# B&R Automation Studio project Soiled_PLC
Automation Studio 4.10.2.37; technology packages: mapp 5.15.0, mappView 5.15.1

## Configuration DisplayCTT11

CPU , AutomationRuntime S3.09, Build 4.1.2, Vc V4.21.1

### Task classes (Cpu.sw)
```
Cyclic#1 (cycle 10000 us, tolerance 10000 us):
  ClientPane <- Displays.ClientPanel.prg
  Client <- Displays.Client.prg
  zzClientTe <- Displays.zzClientText.prg
Cyclic#4 (cycle 100000 us, tolerance 100000 us):
  zzSQLDrive <- SQL.zzSQLDriver.prg
VcDataObjects: CT11 <- Displays.CT11.dob
Binaries: vcdsint, vcctext, arialbd, verdanab, vcalarm, vcshared, vcpdsw, vccline, vcgclass, vccbtn, vcresman, vccnum, vcchspot, vccstr, vccshape, vcfile, Displa03, vcrt, vcbclass, vcfntttf, verdana, vcdsloc, vccovl, arial, Displa02, vcpfmtcx, visvc, Displa, vcmgr, vctcal, vcptelo, vcpdpp30, vcpfpp30, vcpdvnc, vcnet, Displa01, ashwd, sysconf, asfw, arconfig, iomap
Libraries: DispLib, zzSQL_Lib, AsDb, IecCheck, AsString, sys_lib, Ethernet, AsTCP, Visapi, AsARCfg, AsETH, AsIecCon, standard, runtime, astime, fileio, dataobj
```

### Hardware
```
CTT11 : 4PP420.1043-K37 v1.0.1.3
  Connector IF5:
    ActivateDevice = 1
    Mode = Manual
    InternetAddress = 10.8.4.10
    SubnetMask = 255.255.240.0
    Vnc1
    VncVcObjectName1 = CT11
    VncKeyMappingFile1 = VC\PS2-Keyboard.dis
    VncAuthentication1 = 1
    VncPasswordViewOnly1 = 7701
    VncPasswordViewControl1 = medoc
    VncRefreshRate1 = 500
  PermanentPvSize = 17
  RemanentGlobalPvSize = 4300
  VolatileGlobalPvSize = 150000
  PreservePermanentPvMemory = 1
  RebootPowerfail = 2
  Cyclic1Duration = 10000
  Cyclic1Tolerance = 10000
  Cyclic2Duration = 20000
  Cyclic2Tolerance = 20000
  Cyclic3Duration = 50000
  Cyclic3Tolerance = 50000
  Cyclic4Duration = 100000
  Cyclic4Tolerance = 100000
  Cyclic5Duration = 200000
  Cyclic5Tolerance = 200000
  Cyclic6Duration = 500000
  Cyclic6Tolerance = 500000
  Cyclic7Duration = 1000000
  Cyclic7Tolerance = 1000000
  Cyclic8Duration = 10000
  Cyclic8Tolerance = 30000000
  EthernetDefaultGateway = 10.8.15.254
  VcObjectName = CT11
```

### Cpu.per - CTT11/Cpu.per
```iecst
(********************************************************************
 * COPYRIGHT --
 ********************************************************************
 * File: Cpu.per
 * Author: Dave
 * Created: July 20, 2011
 ********************************************************************
 * Declaration of permanent variables
 ********************************************************************)
VAR_CONFIG
	ClientServerIP AT %M0;
END_VAR
```

## Configuration DisplayPCT04

CPU , AutomationRuntime C4.72, Build 4.1.2, Vc V4.72.0

### Task classes (Cpu.sw)
```
Cyclic#1:
  ClientData <- Displays.ClientDataEntry.prg
  ClientPane <- Displays.ClientPanel.prg
  Client <- Displays.Client.prg
  zzClientTe <- Displays.zzClientText.prg
Cyclic#4:
  zzSQLDrive <- SQL.zzSQLDriver.prg
VcDataObjects: PCT04 <- Displays.PCT04.dob
Binaries: vcrt, vcpk, vcfntttf, verdana, vcctext, arial, verdanab, vccovl, vcpfmtcx, vccbtn, vcdsint, vcpdsw, vcpdpp30, vcshared, vcmgr, vcpfpp30, visvc, vcalarm, vcfile, vccnum, vccstr, vcresman, vcgclass, vcdsloc, arialbd, vcptelo, vctcal, vcchspot, vcbclass, vccline, PCT0402, PCT0401, PCT0403, ashwd, sysconf, asfw, iomap, arconfig, vccbmp, Data1, vccshape, vcnet, Data102, Data103, vcpdvnc, Data101
Libraries: DispLib, standard, asieccon, astime, runtime, IecCheck, AsString, sys_lib, astcp, visapi, zzSQL_Lib, AsDb, dataobj, asarcfg, aseth, fileio
```

### Hardware
```
PCT04 : 4PP065.0571-K05 v1.0.2.2
  Connector IF5:
    ActivateDevice = 1
    Mode = Manual
    InternetAddress = 10.8.4.10
    SubnetMask = 255.255.240.0
    Vnc1
    VncVcObjectName1 = PCT04
    VncKeyMappingFile1 = VC\PS2-Keyboard.dis
    VncAuthentication1 = 1
    VncPasswordViewControl1 = medoc
  ConfigurationID = AS4_7_NorthFleetA5_DisplayPCT04
  PermanentPvSize = 17
  RemanentGlobalPvSize = 4300
  VolatileGlobalPvSize = 150000
  EthernetDefaultGateway = 10.8.15.254
  VcObjectName = PCT04
  KeyMappingFile = 4PP065.0571-K05d.dis
```

## Configuration Supertrack

CPU X20CP1586, AutomationRuntime C4.90, Build 4.1.2, Safety 1.10, Vc V4.72.0

### Task classes (Cpu.sw)
```
Cyclic#1 (cycle 1000 us, tolerance 1000 us):
  4_spn1 <- (binary)
  USB_Pmem <- (binary)
  zzClearMem <- (binary)
  can_dry1 <- (binary)
  zzSQLid <- (binary)
  17_svc2 <- (binary)
  18_svc3 <- (binary)
  20_sic3 <- (binary)
  11_spi1 <- (binary)
  17_sp6 <- (binary)
  8_sp8 <- (binary)
  3_svc2 <- (binary)
  2_svc1 <- (binary)
  9_sp6 <- (binary)
  17_sic1 <- (binary)
  8_svc1 <- (binary)
  50_stnsa1 <- (binary)
Cyclic#2 (cycle 10000 us, tolerance 10000 us):
  zzTC2str <- Sequences.10ms.Scan.zzTC2str.prg
  zzGetTime <- Timestamp.zzGetTime.prg
  zzStd <- Sequences.10ms.zzStd.prg
  zzEditBag <- Sequences.10ms.zzEditBag.prg
  zzForceI <- Sequences.10ms.zzForceI.prg
  zzConst <- Sequences.10ms.zzConst.prg
  zzBagID <- Sequences.10ms.zzBagID.prg
  zzTrip <- Sequences.10ms.zzTrip.prg
  zzStnMix <- Sequences.10ms.zzStnMix.prg
  zzBagShuff <- Sequences.10ms.zzBagShuffle.prg
  zzBITcal <- Sequences.10ms.zzBITcal.prg
  zzStnSer <- Sequences.10ms.zzStnSer.prg
  zzcp10ser <- Sequences.10ms.zzcp10ser.prg
  zzStatus <- Sequences.10ms.zzStatus.prg
  zzCusFIFO <- Sequences.10ms.zzCusFIFO.prg
  0_sbelt <- Sequences.10ms.0_sbelt.prg [disabled]
  50_stns1_7 <- Sequences.10ms.50_stns1_7.prg
  50_stn8_14 <- Sequences.10ms.50_stn8_14.prg
  2_stb1B <- Sequences.10ms.2_stb1.prg
  3_clu_1 <- Sequences.10ms.3_clu_1.prg
  4_pn <- Sequences.10ms.4_pn.prg
  5_pf <- Sequences.10ms.5_pf.prg
  6_sdc1 <- Sequences.10ms.6_sdc1.prg
  7_sdc2 <- Sequences.10ms.7_sdc2.prg
  8_sdc3 <- Sequences.10ms.8_sdc3.prg
  9_sdc4 <- Sequences.10ms.9_sdc4.prg
  10_sdc5 <- Sequences.10ms.10_sdc5.prg
  11_sdc6 <- Sequences.10ms.11_sdc6.prg
  12_sdc7 <- Sequences.10ms.12_sdc7.prg
  13_sdc8 <- Sequences.10ms.13_sdc8.prg
  14_sdc9 <- Sequences.10ms.14_sdc9.prg
  15_cbc1 <- Sequences.10ms.15_cbc1.prg
  16_cic1 <- Sequences.10ms.16_cic1.prg
  17_cic2 <- Sequences.10ms.17_cic2.prg
  18_cic3 <- Sequences.10ms.18_cic3.prg
  19_cic4 <- Sequences.10ms.19_cic4.prg
  20_cp1 <- Sequences.10ms.20_cp17.prg
  21_cpi1 <- Sequences.10ms.21_cpi1.prg
  22_cpi2 <- Sequences.10ms.22_cpi2.prg
  23_cpi3 <- Sequences.10ms.23_cpi3.prg
  24_cpi4 <- Sequences.10ms.24_cpi4.prg
  25_cvc1 <- Sequences.10ms.25_cvc1.prg
  26_cp3 <- Sequences.10ms.26_cp3.prg
  27_cp17 <- Sequences.10ms.27_cp17.prg
  28_cp16 <- Sequences.10ms.28_cp16.prg
  29_cp15 <- Sequences.10ms.29_cp15.prg
  30_cp14 <- Sequences.10ms.30_cp14.prg
  31_cp2 <- Sequences.10ms.31_cp2.prg
  32_clu_2 <- Sequences.10ms.3_clu_2.prg
  33_stb2_A <- Sequences.10ms.32_stb2.prg
  34_cpi5 <- Sequences.10ms.34_cpi5.prg
  35_cic5 <- Sequences.10ms.35_cic5.prg
  36_cic6 <- Sequences.10ms.36_cic6.prg
  37_cpi6 <- Sequences.10ms.37_cpi6.prg
  38_cp10 <- Sequences.10ms.38_cp10.prg
  39_cpc1 <- Sequences.10ms.39_cpc1.prg
  40_cp4 <- Sequences.10ms.40_cp4.prg
  41_cp8 <- Sequences.10ms.41_cp8.prg
  42_cp9 <- Sequences.10ms.42_cp9.prg
  43_cp12 <- Sequences.10ms.43_cp12.prg
  44_cpr2 <- Sequences.10ms.44_cpr2.prg
  45_cpr3 <- Sequences.10ms.45_cpr3.prg
  46_cpr4 <- Sequences.10ms.46_cpr4.prg
  47_cpr1 <- Sequences.10ms.47_cpr1.prg
  48_cp6 <- Sequences.10ms.48_cp6.prg
  ssr <- Sequences.10ms.ssr.prg  // speed reducer before SDC2
  zzUld_4 <- Sequences.10ms.zzUld_4.prg
  zzUld_4a <- Sequences.10ms.zzUld_4a.prg [disabled]
  zzForceO <- Sequences.10ms.zzForceO.prg
  zzIndi <- Sequences.10ms.zzIndi.prg [disabled]
  zzTCPIP <- Sequences.10ms.zzTCPIP.prg
  zzIO <- Sequences.10ms.zzIO.prg
  zzOk <- Sequences.10ms.zzOk.prg
  zzDataStor <- Data_BackUp.zzDataStore.prg
  zzTvText <- SQL.zzTvText.prg
  ServerPane <- Displays.ServerPanel.prg
  Server <- Displays.Server.prg
  zzClientTe <- Displays.zzClientText.prg [disabled]
  zzHttpDriv <- http_Lib.zzHttpDriver.prg [disabled]
  zzGetName1 <- SQL.zzGetNamesSQL.zzGetNameSQL.prg [disabled]
  zzTC2end <- Sequences.10ms.Scan.zzTC2end.prg
Cyclic#3:
  zzGetNames <- Sequences.zzGetNames.prg [disabled]
Cyclic#4:
  SafetyUI <- Safety.SafetyUI.prg [disabled]
Cyclic#5:
  HoistServe <- HoistLibrary.HoistServer.prg
  AccessCont <- Safety.AccessControl.prg
  Safety <- Safety.Safety.prg [disabled]
  can_drv1 <- Sequences.200ms.CAN.can_drv1.prg
  can_drv2 <- Sequences.200ms.CAN.can_drv2.prg
  zzWeigh <- Sequences.200ms.zzWeigh.prg
  zzAlarms <- Sequences.200ms.zzAlarms.prg
  zzReport <- Sequences.200ms.Reports.zzReport.prg
  zzStn_Q <- Sequences.200ms.zzStn_Q.prg
  zzTime <- Sequences.200ms.zzTime.prg  // System running time
  CAN_Live <- Sequences.200ms.CAN.CAN_Live.prg
  httpServer <- http_Lib.httpServer.prg [disabled]
Cyclic#8:
  zzModuleLo <- CustomLogs.zzModuleLog.prg
  zzSQLDrive <- SQL.zzSQLDriver.prg [disabled]
  zzWeighSta <- CustomLogs.zzWeighStatus.prg [disabled]
DataObjects: can2_cmd <- Sequences.200ms.CAN.can2_cmd.dob, can1_cmd <- Sequences.200ms.CAN.can1_cmd.dob, arsdmsvp, arsdmhtm, arsdmsvg
Binaries: TCData, udbdef, mvLoader, FWRules, TCLang, iomap, asfw, arconfig, ashwd, sysconf, Role, User, ashwac, TC, OpcUaMap, vcfntttf, vcfile, vcshared, vccshape, vcgclass, arial, CT1102, vcchspot, vcdsint, PCT0403, vccbtn, vcdsloc, vccovl, vccline, vcctext, vcalarm, vcbclass, vcrt, vccnum, vccstr, CT1103, arialbd, PCT0402, vcpdsw, verdanab, verdana, webserv, arsdm
Libraries: ABB_EPL, AsEPL, AsBrMath, AsIOAcc, AsSafety, MTBasics, MTTypes, Ldg_Funct, FileMgr, KanLinkLib, OPCuA, FC302, DataBackUp, standard, runtime, FileIO, Ethernet, dvframe, DataObj, OPERATOR, CAN_Lib, AsTime, AsString, SupLib4, sys_lib, AsTCP, KGstring, AsETH, AsBrStr, AsBrWStr, AsUSB, AsMem, AsArLog, AsUDP, brsystem, AsIODiag, AsARCfg, AsIecCon, IecCheck, AsPciStr, DispLib, zzSQL_Lib, AsDb, KGstdLib, mnParamLib, KL_UserLib, AsHttp, SUP, asxml, ascanopen, arssl, SupFile, vcresman, WETCAN2
```

### Hardware
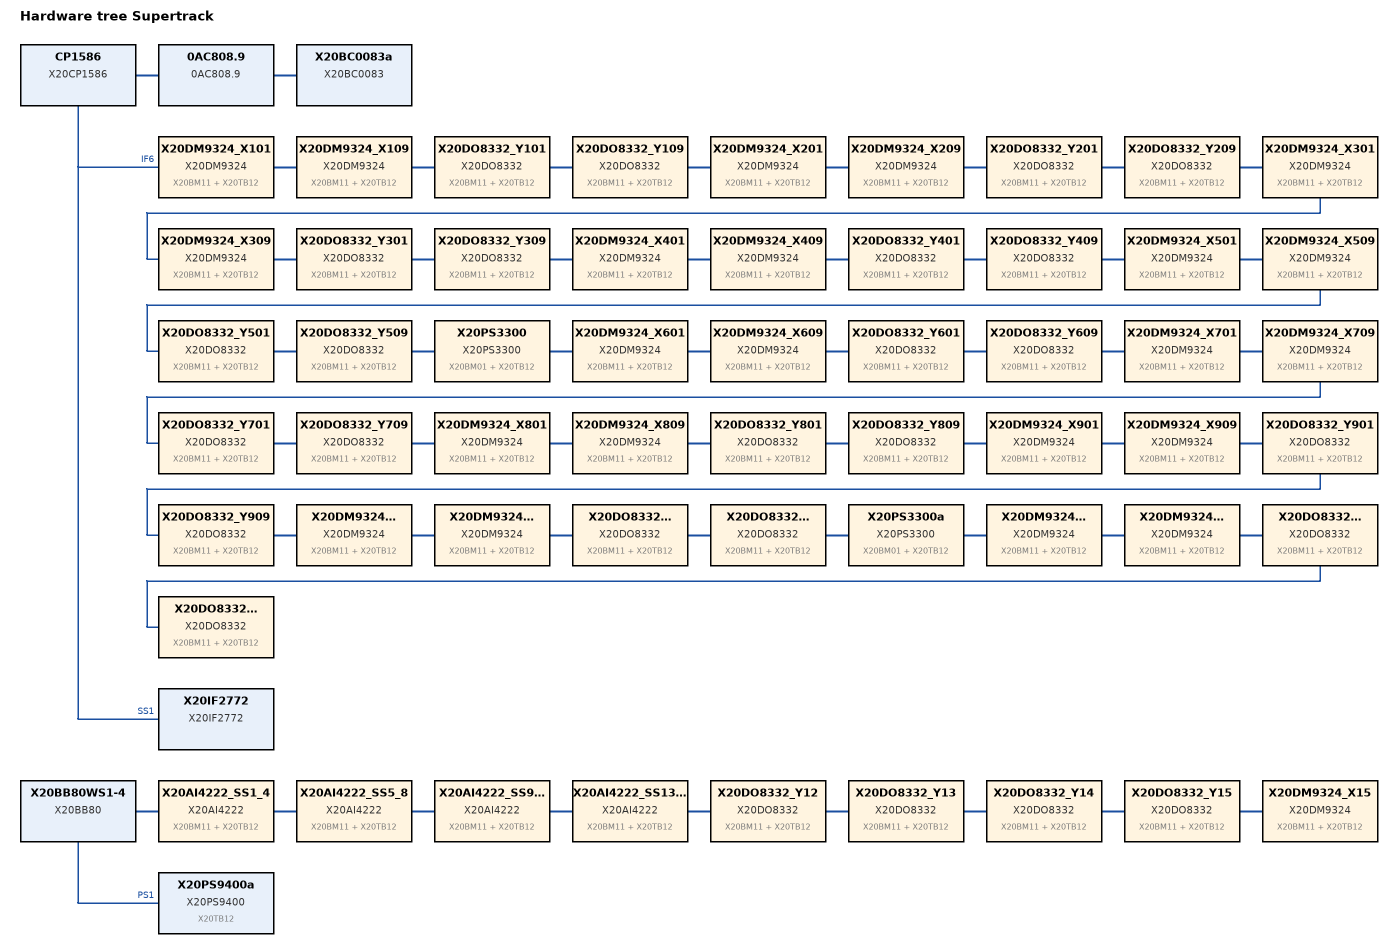
```
0AC808.9 : 0AC808.9 v1.0.0.0  [ETH1 -> CP1586.IF3 [Cable Type=PowerlinkCable, Length=10, Version=1.0.0.3]; ETH8 -> X20BC0083a.PLK1 [Cable Type=PowerlinkCable, Length=10, Version=1.0.0.3]]
CP1586 : X20CP1586 v1.9.0.0
  Connector IF2:
    ActivateDevice = 1
    Baudrate = 100
    Mode = Manual
    InternetAddress = 10.8.4.20
  ConfigurationID = AS4_2_BaseStandard_Supertrack
  UserRamSize = 200000
  RemMemSize = 200000
  PermanentPvSize = 47756
  RemanentGlobalPvSize = 5000
  VolatileGlobalPvSize = 900000
  ClearNvMemoryAfterShutdownFlushError = 0
  CyclicFlushRemMemSelector = 1
  EnableUsbRemoteInstall = 1
  EnableCfRemoteInstall = 1
  Cyclic1Duration = 1000
  Cyclic1Tolerance = 1000
  Cyclic2Duration = 10000
  Cyclic2Tolerance = 10000
  FileDevice1
  FileDeviceName1 = USBStick
  FileDevicePath1 = /bd0\
  ActivateDaylightSavingTime = 1
  ActivateSntp = 1
  SntpcServAddr1 = 10.8.15.254
  EthernetHostName = SupertrackPLC
  EthernetDefaultGateway = 10.8.15.254
  FtpUser1
  FtpUsername1 = admin
  FtpUserPassword1 = vwQCGOhDKwuFhUdMhisKVJgiKzmoNTQazzJQnTTJsZU=  // admin
  FtpUserSalt1 = XFuy8Eo/
  FTPAccessRight1 = 0
  ActivateOpcUa = 1
  OpcUa_AuthenticationTokenType_EnableAnonymous = 0
  OpcUaInformationModels_PV_Version = 1
X20AI4222_SS13_14 : X20AI4222 v1.1.0.0  [SS1 -> X20TB12aq.SS; SL -> X20BM11am.SL1]
  Supervision = off
X20AI4222_SS1_4 : X20AI4222 v1.1.0.0  [SS1 -> X20TB12as.SS; SL -> X20BM11ak.SL1]
  Supervision = off
X20AI4222_SS5_8 : X20AI4222 v1.1.0.0  [SS1 -> X20TB12n.SS; SL -> X20BM11ao.SL1]
  Supervision = off
X20AI4222_SS9_12 : X20AI4222 v1.1.0.0  [SS1 -> X20TB12aw.SS; SL -> X20BM11av.SL1]
  Supervision = off
X20BB80WS1-4 : X20BB80 v1.1.0.0
X20BC0083a : X20BC0083 v2.14.0.0  [PLK1 -> 0AC808.9.ETH8 (NodeNumber=2) [Cable Type=PowerlinkCable, Length=10, Version=1.0.0.3]; SL -> X20BB80WS1-4.SL1]
  Supervision = off
X20BM01 : X20BM01 v2.2.0.0  [X2X1 -> X20BM11s.X2X2]
X20BM01a : X20BM01 v2.2.0.0  [X2X1 -> X20BM11aj.X2X2]
X20BM11 : X20BM11 v1.1.0.0  [X2X1 -> CP1586.IF6]
X20BM11a : X20BM11 v1.1.0.0  [X2X1 -> X20BM11.X2X2]
X20BM11aa : X20BM11 v1.1.0.0  [X2X1 -> X20BM11z.X2X2]
X20BM11ab : X20BM11 v1.1.0.0  [X2X1 -> X20BM11aa.X2X2]
X20BM11ac : X20BM11 v1.1.0.0  [X2X1 -> X20BM11ab.X2X2]
X20BM11ad : X20BM11 v1.1.0.0  [X2X1 -> X20BM11ac.X2X2]
X20BM11ae : X20BM11 v1.1.0.0  [X2X1 -> X20BM11ad.X2X2]
X20BM11af : X20BM11 v1.1.0.0  [X2X1 -> X20BM11ag.X2X2]
X20BM11ag : X20BM11 v1.1.0.0  [X2X1 -> X20BM11as.X2X2]
X20BM11ah : X20BM11 v1.1.0.0  [X2X1 -> X20BM11at.X2X2]
X20BM11ai : X20BM11 v1.1.0.0  [X2X1 -> X20BM11au.X2X2]
X20BM11aj : X20BM11 v1.1.0.0  [X2X1 -> X20BM11ai.X2X2]
X20BM11ak : X20BM11 v1.1.0.0  [X2X1 -> X20BB80WS1-4.IF1]
X20BM11al : X20BM11 v1.1.0.0  [X2X1 -> X20BM11an.X2X2]
X20BM11am : X20BM11 v1.1.0.0  [X2X1 -> X20BM11av.X2X2]
X20BM11an : X20BM11 v1.1.0.0  [X2X1 -> X20BM11bc.X2X2]
X20BM11ao : X20BM11 v1.1.0.0  [X2X1 -> X20BM11ak.X2X2]
X20BM11as : X20BM11 v1.1.0.0  [X2X1 -> X20BM11ae.X2X2]
X20BM11at : X20BM11 v1.1.0.0  [X2X1 -> X20BM11af.X2X2]
X20BM11au : X20BM11 v1.1.0.0  [X2X1 -> X20BM11ah.X2X2]
X20BM11av : X20BM11 v1.1.0.0  [X2X1 -> X20BM11ao.X2X2]
X20BM11aw : X20BM11 v1.1.0.0  [X2X1 -> X20BM11am.X2X2]
X20BM11ax : X20BM11 v1.1.0.0  [X2X1 -> X20BM01a.X2X2]
X20BM11ay : X20BM11 v1.1.0.0  [X2X1 -> X20BM11ax.X2X2]
X20BM11az : X20BM11 v1.1.0.0  [X2X1 -> X20BM11ay.X2X2]
X20BM11b : X20BM11 v1.1.0.0  [X2X1 -> X20BM11a.X2X2]
X20BM11ba : X20BM11 v1.1.0.0  [X2X1 -> X20BM11az.X2X2]
X20BM11bb : X20BM11 v1.1.0.0  [X2X1 -> X20BM11aw.X2X2]
X20BM11bc : X20BM11 v1.1.0.0  [X2X1 -> X20BM11bb.X2X2]
X20BM11c : X20BM11 v1.1.0.0  [X2X1 -> X20BM11b.X2X2]
X20BM11d : X20BM11 v1.1.0.0  [X2X1 -> X20BM11c.X2X2]
X20BM11e : X20BM11 v1.1.0.0  [X2X1 -> X20BM11d.X2X2]
X20BM11f : X20BM11 v1.1.0.0  [X2X1 -> X20BM11e.X2X2]
X20BM11g : X20BM11 v1.1.0.0  [X2X1 -> X20BM11f.X2X2]
X20BM11h : X20BM11 v1.1.0.0  [X2X1 -> X20BM11g.X2X2]
X20BM11i : X20BM11 v1.1.0.0  [X2X1 -> X20BM11h.X2X2]
X20BM11j : X20BM11 v1.1.0.0  [X2X1 -> X20BM11i.X2X2]
X20BM11k : X20BM11 v1.1.0.0  [X2X1 -> X20BM11j.X2X2]
X20BM11l : X20BM11 v1.1.0.0  [X2X1 -> X20BM11k.X2X2]
X20BM11m : X20BM11 v1.1.0.0  [X2X1 -> X20BM11l.X2X2]
X20BM11n : X20BM11 v1.1.0.0  [X2X1 -> X20BM11m.X2X2]
X20BM11o : X20BM11 v1.1.0.0  [X2X1 -> X20BM11n.X2X2]
X20BM11p : X20BM11 v1.1.0.0  [X2X1 -> X20BM11o.X2X2]
X20BM11q : X20BM11 v1.1.0.0  [X2X1 -> X20BM11p.X2X2]
X20BM11r : X20BM11 v1.1.0.0  [X2X1 -> X20BM11q.X2X2]
X20BM11s : X20BM11 v1.1.0.0  [X2X1 -> X20BM11r.X2X2]
X20BM11t : X20BM11 v1.1.0.0  [X2X1 -> X20BM01.X2X2]
X20BM11u : X20BM11 v1.1.0.0  [X2X1 -> X20BM11t.X2X2]
X20BM11v : X20BM11 v1.1.0.0  [X2X1 -> X20BM11u.X2X2]
X20BM11w : X20BM11 v1.1.0.0  [X2X1 -> X20BM11v.X2X2]
X20BM11x : X20BM11 v1.1.0.0  [X2X1 -> X20BM11w.X2X2]
X20BM11y : X20BM11 v1.1.0.0  [X2X1 -> X20BM11x.X2X2]
X20BM11z : X20BM11 v1.1.0.0  [X2X1 -> X20BM11y.X2X2]
X20DM9324_X1001 : X20DM9324 v1.2.0.0  [SS1 -> X20TB12ak.SS; SL -> X20BM11ah.SL1]
  Supervision = off
X20DM9324_X1009 : X20DM9324 v1.2.0.0  [SS1 -> X20TB12ba.SS; SL -> X20BM11au.SL1]
  Supervision = off
X20DM9324_X101 : X20DM9324 v1.2.0.0  [SS1 -> X20TB12.SS; SL -> X20BM11.SL1]
  Supervision = off
X20DM9324_X109 : X20DM9324 v1.2.0.0  [SS1 -> X20TB12a.SS; SL -> X20BM11a.SL1]
  Supervision = off
X20DM9324_X1101 : X20DM9324 v1.2.0.0  [SS1 -> X20TB12bd.SS; SL -> X20BM11ax.SL1]
  Supervision = off
X20DM9324_X1109 : X20DM9324 v1.2.0.0  [SS1 -> X20TB12be.SS; SL -> X20BM11ay.SL1]
  Supervision = off
X20DM9324_X15 : X20DM9324 v1.2.0.0  [SS1 -> X20TB12ap.SS; SL -> X20BM11al.SL1]
  Supervision = off
X20DM9324_X201 : X20DM9324 v1.2.0.0  [SS1 -> X20TB12d.SS; SL -> X20BM11d.SL1]
  Supervision = off
X20DM9324_X209 : X20DM9324 v1.2.0.0  [SS1 -> X20TB12e.SS; SL -> X20BM11e.SL1]
  Supervision = off
X20DM9324_X301 : X20DM9324 v1.2.0.0  [SS1 -> X20TB12h.SS; SL -> X20BM11h.SL1]
  Supervision = off
X20DM9324_X309 : X20DM9324 v1.2.0.0  [SS1 -> X20TB12i.SS; SL -> X20BM11i.SL1]
  Supervision = off
X20DM9324_X401 : X20DM9324 v1.2.0.0  [SS1 -> X20TB12l.SS; SL -> X20BM11l.SL1]
  Supervision = off
X20DM9324_X409 : X20DM9324 v1.2.0.0  [SS1 -> X20TB12m.SS; SL -> X20BM11m.SL1]
  Supervision = off
X20DM9324_X501 : X20DM9324 v1.2.0.0  [SS1 -> X20TB12q.SS; SL -> X20BM11p.SL1]
  Supervision = off
X20DM9324_X509 : X20DM9324 v1.2.0.0  [SS1 -> X20TB12r.SS; SL -> X20BM11q.SL1]
  Supervision = off
X20DM9324_X601 : X20DM9324 v1.2.0.0  [SS1 -> X20TB12v.SS; SL -> X20BM11t.SL1]
  Supervision = off
X20DM9324_X609 : X20DM9324 v1.2.0.0  [SS1 -> X20TB12w.SS; SL -> X20BM11u.SL1]
  Supervision = off
X20DM9324_X701 : X20DM9324 v1.2.0.0  [SS1 -> X20TB12z.SS; SL -> X20BM11x.SL1]
  Supervision = off
X20DM9324_X709 : X20DM9324 v1.2.0.0  [SS1 -> X20TB12aa.SS; SL -> X20BM11y.SL1]
  Supervision = off
X20DM9324_X801 : X20DM9324 v1.2.0.0  [SS1 -> X20TB12ad.SS; SL -> X20BM11ab.SL1]
  Supervision = off
X20DM9324_X809 : X20DM9324 v1.2.0.0  [SS1 -> X20TB12ae.SS; SL -> X20BM11ac.SL1]
  Supervision = off
X20DM9324_X901 : X20DM9324 v1.2.0.0  [SS1 -> X20TB12ah.SS; SL -> X20BM11as.SL1]
  Supervision = off
X20DM9324_X909 : X20DM9324 v1.2.0.0  [SS1 -> X20TB12aj.SS; SL -> X20BM11ag.SL1]
  Supervision = off
X20DO8332_Y1001 : X20DO8332 v1.5.0.0  [SS1 -> X20TB12al.SS; SL -> X20BM11ai.SL1]
  Supervision = off
X20DO8332_Y1009 : X20DO8332 v1.5.0.0  [SS1 -> X20TB12am.SS; SL -> X20BM11aj.SL1]
  Supervision = off
X20DO8332_Y101 : X20DO8332 v1.5.0.0  [SS1 -> X20TB12b.SS; SL -> X20BM11b.SL1]
  Supervision = off
X20DO8332_Y109 : X20DO8332 v1.5.0.0  [SS1 -> X20TB12c.SS; SL -> X20BM11c.SL1]
  Supervision = off
X20DO8332_Y1101 : X20DO8332 v1.5.0.0  [SS1 -> X20TB12bf.SS; SL -> X20BM11az.SL1]
  Supervision = off
X20DO8332_Y1109 : X20DO8332 v1.5.0.0  [SS1 -> X20TB12bg.SS; SL -> X20BM11ba.SL1]
  Supervision = off
X20DO8332_Y12 : X20DO8332 v1.5.0.0  [SS1 -> X20TB12bb.SS; SL -> X20BM11aw.SL1]
  Supervision = off
X20DO8332_Y13 : X20DO8332 v1.5.0.0  [SS1 -> X20TB12bc.SS; SL -> X20BM11bb.SL1]
  Supervision = off
X20DO8332_Y14 : X20DO8332 v1.5.0.0  [SS1 -> X20TB12bh.SS; SL -> X20BM11bc.SL1]
  Supervision = off
X20DO8332_Y15 : X20DO8332 v1.5.0.0  [SS1 -> X20TB12ar.SS; SL -> X20BM11an.SL1]
  Supervision = off
X20DO8332_Y201 : X20DO8332 v1.5.0.0  [SS1 -> X20TB12f.SS; SL -> X20BM11f.SL1]
  Supervision = off
X20DO8332_Y209 : X20DO8332 v1.5.0.0  [SS1 -> X20TB12g.SS; SL -> X20BM11g.SL1]
  Supervision = off
X20DO8332_Y301 : X20DO8332 v1.5.0.0  [SS1 -> X20TB12j.SS; SL -> X20BM11j.SL1]
  Supervision = off
X20DO8332_Y309 : X20DO8332 v1.5.0.0  [SS1 -> X20TB12k.SS; SL -> X20BM11k.SL1]
  Supervision = off
X20DO8332_Y401 : X20DO8332 v1.5.0.0  [SS1 -> X20TB12o.SS; SL -> X20BM11n.SL1]
  Supervision = off
X20DO8332_Y409 : X20DO8332 v1.5.0.0  [SS1 -> X20TB12p.SS; SL -> X20BM11o.SL1]
  Supervision = off
X20DO8332_Y501 : X20DO8332 v1.5.0.0  [SS1 -> X20TB12s.SS; SL -> X20BM11r.SL1]
  Supervision = off
X20DO8332_Y509 : X20DO8332 v1.5.0.0  [SS1 -> X20TB12t.SS; SL -> X20BM11s.SL1]
  Supervision = off
X20DO8332_Y601 : X20DO8332 v1.5.0.0  [SS1 -> X20TB12x.SS; SL -> X20BM11v.SL1]
  Supervision = off
X20DO8332_Y609 : X20DO8332 v1.5.0.0  [SS1 -> X20TB12y.SS; SL -> X20BM11w.SL1]
  Supervision = off
X20DO8332_Y701 : X20DO8332 v1.5.0.0  [SS1 -> X20TB12ab.SS; SL -> X20BM11z.SL1]
  Supervision = off
X20DO8332_Y709 : X20DO8332 v1.5.0.0  [SS1 -> X20TB12ac.SS; SL -> X20BM11aa.SL1]
  Supervision = off
X20DO8332_Y801 : X20DO8332 v1.5.0.0  [SS1 -> X20TB12af.SS; SL -> X20BM11ad.SL1]
  Supervision = off
X20DO8332_Y809 : X20DO8332 v1.5.0.0  [SS1 -> X20TB12ag.SS; SL -> X20BM11ae.SL1]
  Supervision = off
X20DO8332_Y901 : X20DO8332 v1.5.0.0  [SS1 -> X20TB12ai.SS; SL -> X20BM11af.SL1]
  Supervision = off
X20DO8332_Y909 : X20DO8332 v1.5.0.0  [SS1 -> X20TB12az.SS; SL -> X20BM11at.SL1]
  Supervision = off
X20IF2772 : X20IF2772 v1.5.0.0  [SS -> CP1586.SS1]
X20PS3300 : X20PS3300 v1.3.0.0  [SS1 -> X20TB12u.SS; SL -> X20BM01.SL1]
  Supervision = off
X20PS3300a : X20PS3300 v1.3.0.0  [SS1 -> X20TB12an.SS; SL -> X20BM01a.SL1]
  Supervision = off
X20PS9400a : X20PS9400 v1.7.0.0  [SS1 -> X20TB12ao.SS; PS -> X20BB80WS1-4.PS1]
  Supervision = off
X20TB12 : X20TB12 v1.0.0.0
X20TB12a : X20TB12 v1.0.0.0
X20TB12aa : X20TB12 v1.0.0.0
X20TB12ab : X20TB12 v1.0.0.0
X20TB12ac : X20TB12 v1.0.0.0
X20TB12ad : X20TB12 v1.0.0.0
X20TB12ae : X20TB12 v1.0.0.0
X20TB12af : X20TB12 v1.0.0.0
X20TB12ag : X20TB12 v1.0.0.0
X20TB12ah : X20TB12 v1.0.0.0
X20TB12ai : X20TB12 v1.0.0.0
X20TB12aj : X20TB12 v1.0.0.0
X20TB12ak : X20TB12 v1.0.0.0
X20TB12al : X20TB12 v1.0.0.0
X20TB12am : X20TB12 v1.0.0.0
X20TB12an : X20TB12 v1.0.0.0
X20TB12ao : X20TB12 v1.0.0.0
X20TB12ap : X20TB12 v1.0.0.0
X20TB12aq : X20TB12 v1.0.0.0
X20TB12ar : X20TB12 v1.0.0.0
X20TB12as : X20TB12 v1.0.0.0
X20TB12aw : X20TB12 v1.0.0.0
X20TB12az : X20TB12 v1.0.0.0
X20TB12b : X20TB12 v1.0.0.0
X20TB12ba : X20TB12 v1.0.0.0
X20TB12bb : X20TB12 v1.0.0.0
X20TB12bc : X20TB12 v1.0.0.0
X20TB12bd : X20TB12 v1.0.0.0
X20TB12be : X20TB12 v1.0.0.0
X20TB12bf : X20TB12 v1.0.0.0
X20TB12bg : X20TB12 v1.0.0.0
X20TB12bh : X20TB12 v1.0.0.0
X20TB12c : X20TB12 v1.0.0.0
X20TB12d : X20TB12 v1.0.0.0
X20TB12e : X20TB12 v1.0.0.0
X20TB12f : X20TB12 v1.0.0.0
X20TB12g : X20TB12 v1.0.0.0
X20TB12h : X20TB12 v1.0.0.0
X20TB12i : X20TB12 v1.0.0.0
X20TB12j : X20TB12 v1.0.0.0
X20TB12k : X20TB12 v1.0.0.0
X20TB12l : X20TB12 v1.0.0.0
X20TB12m : X20TB12 v1.0.0.0
X20TB12n : X20TB12 v1.0.0.0
X20TB12o : X20TB12 v1.0.0.0
X20TB12p : X20TB12 v1.0.0.0
X20TB12q : X20TB12 v1.0.0.0
X20TB12r : X20TB12 v1.0.0.0
X20TB12s : X20TB12 v1.0.0.0
X20TB12t : X20TB12 v1.0.0.0
X20TB12u : X20TB12 v1.0.0.0
X20TB12v : X20TB12 v1.0.0.0
X20TB12w : X20TB12 v1.0.0.0
X20TB12x : X20TB12 v1.0.0.0
X20TB12y : X20TB12 v1.0.0.0
X20TB12z : X20TB12 v1.0.0.0
```

### 230104.iom - CP1586/230104.iom
```iecst
08:04:57, Error= -2147217873,  CmdExport  [Microsoft][ODBC Microsoft Access Driver] The changes you requested to the table were not successful because they would create duplicate values in the index, primary key, or relationship.  Change the data in the field or fields that contain duplicate data, remove the index, or redefine the index to permit duplicate entries and try again.
```

### 230121.iom - CP1586/230121.iom
```iecst
16:15:44, Error= -2147217873,  CmdExport  [Microsoft][ODBC Microsoft Access Driver] The changes you requested to the table were not successful because they would create duplicate values in the index, primary key, or relationship.  Change the data in the field or fields that contain duplicate data, remove the index, or redefine the index to permit duplicate entries and try again.
```

### Cpu.per - CP1586/Cpu.per
```iecst
(********************************************************************
 * COPYRIGHT --
 ********************************************************************
 * File: Cpu.per
 * Author: Dave
 * Created: November 19, 2010
 ********************************************************************
 * Declaration of permanent variables
 ********************************************************************)
VAR_CONFIG
	C AT %MW0; (* *)
	D AT %MW200; (* *)
	D32 AT %MD16200; (* *)
	RB_Posn AT %M20200; (* *)
	RB_Perm AT %M22632; (* *)
	SQL AT %M22696; (* *)
	ReportBuffer AT %M22956; (* *)
	Bag AT %M31756; (* *)
END_VAR
```

### IoMap.iom - CP1586/IoMap.iom
```iecst
(********************************************************************
 * COPYRIGHT --
 ********************************************************************
 * File: IoMap.iom
 * Author: Dave
 * Created: November 19, 2010
 ********************************************************************
 * IO mapping file
 ********************************************************************)
VAR_CONFIG
	OK[1] AT %IX."X20DM9324_X101".ModuleOk;
	X[1].X01 AT %IX."X20DM9324_X101".DigitalInput01; (*CDC 5 Bag at buffer   *)
	X[1].X02 AT %IX."X20DM9324_X101".DigitalInput02; (*CDC 5 Bag at buffer stop *)
	X[1].X03 AT %IX."X20DM9324_X101".DigitalInput03; (*CDC 5 Bag in discharger*)
	X[1].X04 AT %IX."X20DM9324_X101".DigitalInput04; (*CDC 5 Bag out of discharger *)
	X[1].X05 AT %IX."X20DM9324_X101".DigitalInput05; (*CDC 5 Drop load *)
	X[1].X06 AT %IX."X20DM9324_X101".DigitalInput06; (*CDC 5 Load dropped *)
	X[1].X07 AT %IX."X20DM9324_X101".DigitalInput07; (*CDC 6 Bag at buffer *)
	X[1].X08 AT %IX."X20DM9324_X101".DigitalInput08; (*CDC 6 Bag at buffer stop *)
	OK[2] AT %IX."X20DM9324_X109".ModuleOk;
	X[1].X09 AT %IX."X20DM9324_X109".DigitalInput01; (*CDC 6 Bag in discharger  *)
	X[1].X10 AT %IX."X20DM9324_X109".DigitalInput02; (*CDC 6 Bag out of discharger *)
	X[1].X11 AT %IX."X20DM9324_X109".DigitalInput03; (*CDC 6 Drop load *)
	X[1].X12 AT %IX."X20DM9324_X109".DigitalInput04; (*CDC 6 Load dropped  *)
	X[1].X13 AT %IX."X20DM9324_X109".DigitalInput05; (*CDC 7 Bag at buffer  *)
	X[1].X14 AT %IX."X20DM9324_X109".DigitalInput06; (*CDC 7 Bag at buffer stop *)
	X[1].X15 AT %IX."X20DM9324_X109".DigitalInput07; (*CDC 7 Bag in discharger *)
	X[1].X16 AT %IX."X20DM9324_X109".DigitalInput08; (*CDC 7 Bag out of discharger  *)
	OK[3] AT %IX."X20DO8332_Y101".ModuleOk;
	Y[1].Y01 AT %QX."X20DO8332_Y101".DigitalOutput01; (*CP 10 Select point to SDC 5 *)
	Y[1].Y02 AT %QX."X20DO8332_Y101".DigitalOutput02; (*CDC 5 Open buffer stop *)
	Y[1].Y03 AT %QX."X20DO8332_Y101".DigitalOutput03; (*CDC 5 Open discharger stop *)
	Y[1].Y04 AT %QX."X20DO8332_Y101".DigitalOutput04; (*CDC 5 Steady cylinders *)
	Y[1].Y05 AT %QX."X20DO8332_Y101".DigitalOutput05; (*CDC 5 Bag ready *)
	Y[1].Y06 AT %QX."X20DO8332_Y101".DigitalOutput06; (*CDC 5 Open bag *)
	Y[1].Y07 AT %QX."X20DO8332_Y101".DigitalOutput07; (*CP 11 Select point to SDC 6 *)
	Y[1].Y08 AT %QX."X20DO8332_Y101".DigitalOutput08; (*CDC 6 Open buffer stop *)
	OK[4] AT %IX."X20DO8332_Y109".ModuleOk;
	Y[1].Y09 AT %QX."X20DO8332_Y109".DigitalOutput01; (*CDC 6 Open discharger stop + CP 14*)
	Y[1].Y10 AT %QX."X20DO8332_Y109".DigitalOutput02; (*CDC 6 Steady cylinders*)
	Y[1].Y11 AT %QX."X20DO8332_Y109".DigitalOutput03; (*CDC 6 Bag ready *)
	Y[1].Y12 AT %QX."X20DO8332_Y109".DigitalOutput04; (*CDC 6 Open bag*)
	Y[1].Y13 AT %QX."X20DO8332_Y109".DigitalOutput05; (*CP 12 Select point to SDC 7 *)
	Y[1].Y14 AT %QX."X20DO8332_Y109".DigitalOutput06; (*CDC 7 Open buffer stop *)
	Y[1].Y15 AT %QX."X20DO8332_Y109".DigitalOutput07; (*CDC 7 Open discharger stop + CP 15*)
	Y[1].Y16 AT %QX."X20DO8332_Y109".DigitalOutput08; (*CDC 7 Steady cylinders *)
	OK[5] AT %IX."X20DM9324_X201".ModuleOk;
	X[2].X01 AT %IX."X20DM9324_X201".DigitalInput01; (*CDC 7 Drop load    *)
	X[2].X02 AT %IX."X20DM9324_X201".DigitalInput02; (*CDC 7 Load dropped *)
	X[2].X03 AT %IX."X20DM9324_X201".DigitalInput03; (*CDC 8 Bag at buffer *)
	X[2].X04 AT %IX."X20DM9324_X201".DigitalInput04; (*CDC 8 Bag at buffer stop *)
	X[2].X05 AT %IX."X20DM9324_X201".DigitalInput05; (*CDC 8 Bag in discharger *)
	X[2].X06 AT %IX."X20DM9324_X201".DigitalInput06; (*CDC 8 Bag out of discharger*)
	X[2].X07 AT %IX."X20DM9324_X201".DigitalInput07; (*CDC 8 Drop load *)
	X[2].X08 AT %IX."X20DM9324_X201".DigitalInput08; (*CDC 8 Load dropped *)
	OK[6] AT %IX."X20DM9324_X209".ModuleOk;
	X[2].X09 AT %IX."X20DM9324_X209".DigitalInput01; (*CDC9 Bag at buffer*)
	X[2].X10 AT %IX."X20DM9324_X209".DigitalInput02; (*CDC 9 Bag at buffer stop *)
	X[2].X11 AT %IX."X20DM9324_X209".DigitalInput03; (*CDC 9 Bag in discharger *)
	X[2].X12 AT %IX."X20DM9324_X209".DigitalInput04; (*CDC 9 Bag out of discharger *)
	X[2].X13 AT %IX."X20DM9324_X209".DigitalInput05; (*CDC 9 Drop load *)
	X[2].X14 AT %IX."X20DM9324_X209".DigitalInput06; (*CDC 9 Load dropped *)
	X[2].X15 AT %IX."X20DM9324_X209".DigitalInput07; (*Spare *)
	X[2].X16 AT %IX."X20DM9324_X209".DigitalInput08; (*CIC 6 Bag at buffer stop *)
	OK[7] AT %IX."X20DO8332_Y201".ModuleOk;
	Y[2].Y01 AT %QX."X20DO8332_Y201".DigitalOutput01; (*CDC 7 Bag ready*)
	Y[2].Y02 AT %QX."X20DO8332_Y201".DigitalOutput02; (*CDC 7 Open bag*)
	Y[2].Y03 AT %QX."X20DO8332_Y201".DigitalOutput03; (*CP13 Select CDC8*)
	Y[2].Y04 AT %QX."X20DO8332_Y201".DigitalOutput04; (*CDC 8 Open buffer stop*)
	Y[2].Y05 AT %QX."X20DO8332_Y201".DigitalOutput05; (*CDC 8 Open discharger stop + CP 16*)
	Y[2].Y06 AT %QX."X20DO8332_Y201".DigitalOutput06; (*CDC 8 Steady cylinders *)
	Y[2].Y07 AT %QX."X20DO8332_Y201".DigitalOutput07; (*CDC 8 Bag ready*)
	Y[2].Y08 AT %QX."X20DO8332_Y201".DigitalOutput08; (*CDC 8 Open bag*)
	OK[8] AT %IX."X20DO8332_Y209".ModuleOk;
	Y[2].Y09 AT %QX."X20DO8332_Y209".DigitalOutput01; (*Spare*)
	Y[2].Y10 AT %QX."X20DO8332_Y209".DigitalOutput02; (*CDC 9 Open buffer stop*)
	Y[2].Y11 AT %QX."X20DO8332_Y209".DigitalOutput03; (*CDC 9 Open discharger stop + CP 17*)
	Y[2].Y12 AT %QX."X20DO8332_Y209".DigitalOutput04; (*CDC 9 Steady cylinders*)
	Y[2].Y13 AT %QX."X20DO8332_Y209".DigitalOutput05; (*CDC 9 Bag ready*)
	Y[2].Y14 AT %QX."X20DO8332_Y209".DigitalOutput06; (*CDC 9 Open bag*)
	Y[2].Y15 AT %QX."X20DO8332_Y209".DigitalOutput07; (*CIC 5 Open buffer stop*)
	Y[2].Y16 AT %QX."X20DO8332_Y209".DigitalOutput08; (*CIC 6 Open buffer stop*)
	OK[9] AT %IX."X20DM9324_X301".ModuleOk;
	X[3].X01 AT %IX."X20DM9324_X301".DigitalInput01; (*Alarm Cancel *)
	X[3].X02 AT %IX."X20DM9324_X301".DigitalInput02; (*Sorting belt A photocell*)
	X[3].X03 AT %IX."X20DM9324_X301".DigitalInput03; (*CLU1 Bag at buffer stop*)
	X[3].X04 AT %IX."X20DM9324_X301".DigitalInput04; (*CLU1 Bag passed stop*)
	X[3].X05 AT %IX."X20DM9324_X301".DigitalInput05; (*CLU1 Bag at loading unit stop*)
	X[3].X06 AT %IX."X20DM9324_X301".DigitalInput06; (*CLU 1 Bag out of loading unit*)
	X[3].X07 AT %IX."X20DM9324_X301".DigitalInput07; (*Sorting belt B photocell*)
	X[3].X08 AT %IX."X20DM9324_X301".DigitalInput08; (*CLU2 Bag at buffer stop*)
	OK[10] AT %IX."X20DM9324_X309".ModuleOk;
	X[3].X09 AT %IX."X20DM9324_X309".DigitalInput01; (*CLU2 Bag passed stop*)
	X[3].X10 AT %IX."X20DM9324_X309".DigitalInput02; (*CLU2 Bag at loading unit stop*)
	X[3].X11 AT %IX."X20DM9324_X309".DigitalInput03; (*CLU2 Bag out of loading unit*)
	X[3].X12 AT %IX."X20DM9324_X309".DigitalInput04; (*Bag at CVC1 buffer*)
	X[3].X13 AT %IX."X20DM9324_X309".DigitalInput05; (*CVC1 Bag at low level buffer stop*)
	X[3].X14 AT %IX."X20DM9324_X309".DigitalInput06; (*CVC1 Carriage at bottom*)
	X[3].X15 AT %IX."X20DM9324_X309".DigitalInput07; (*CVC1 Carriage at top*)
	X[3].X16 AT %IX."X20DM9324_X309".DigitalInput08; (*CVC1 Bag out at top*)
	OK[11] AT %IX."X20DO8332_Y301".ModuleOk;
	Y[3].Y01 AT %QX."X20DO8332_Y301".DigitalOutput01; (*Alarm Output*)
	Y[3].Y02 AT %QX."X20DO8332_Y301".DigitalOutput02; (*CLU1 Buffer stop*)
	Y[3].Y03 AT %QX."X20DO8332_Y301".DigitalOutput03; (*CLU1 Elephants foot*)
	Y[3].Y04 AT %QX."X20DO8332_Y301".DigitalOutput04; (*CLU1 Steady cylinder*)
	Y[3].Y05 AT %QX."X20DO8332_Y301".DigitalOutput05; (*CLU1 Loading unit stop*)
	Y[3].Y06 AT %QX."X20DO8332_Y301".DigitalOutput06; (*CLU2 Buffer stop*)
	Y[3].Y07 AT %QX."X20DO8332_Y301".DigitalOutput07; (*Spare*)
	Y[3].Y08 AT %QX."X20DO8332_Y301".DigitalOutput08; (*CLU2 Steady cylinder*)
	OK[12] AT %IX."X20DO8332_Y309".ModuleOk;
	Y[3].Y09 AT %QX."X20DO8332_Y309".DigitalOutput01; (*CLU2 Loading unit stop*)
	Y[3].Y10 AT %QX."X20DO8332_Y309".DigitalOutput02; (*Select CP1 from CLU1*)
	Y[3].Y11 AT %QX."X20DO8332_Y309".DigitalOutput03; (*Select CP1 from CLU2*)
	Y[3].Y12 AT %QX."X20DO8332_Y309".DigitalOutput04; (*CVC 1 Low level buffer stop*)
	Y[3].Y13 AT %QX."X20DO8332_Y309".DigitalOutput05; (*CPI 1 Buffer stop*)
	Y[3].Y14 AT %QX."X20DO8332_Y309".DigitalOutput06; (*CPI 2 Buffer stop*)
	Y[3].Y15 AT %QX."X20DO8332_Y309".DigitalOutput07; (*CPI 3 Buffer stop*)
	Y[3].Y16 AT %QX."X20DO8332_Y309".DigitalOutput08; (*CPI 4 Buffer stop*)
	OK[13] AT %IX."X20DM9324_X401".ModuleOk;
	X[4].X01 AT %IX."X20DM9324_X401".DigitalInput01; (*Ongoing bag arrived line 1*)
	X[4].X02 AT %IX."X20DM9324_X401".DigitalInput02; (*Ongoing bag arrived line 2*)
	X[4].X03 AT %IX."X20DM9324_X401".DigitalInput03; (*Ongoing bag arrived line 3*)
	X[4].X04 AT %IX."X20DM9324_X401".DigitalInput04; (*Ongoing bag arrived line 4*)
	X[4].X05 AT %IX."X20DM9324_X401".DigitalInput05; (*Ongoing bag arrived line 5*)
	X[4].X06 AT %IX."X20DM9324_X401".DigitalInput06; (*Ongoing bag arrived line 6*)
	X[4].X07 AT %IX."X20DM9324_X401".DigitalInput07; (*CSR 1 Speed reducor 1*)
	X[4].X08 AT %IX."X20DM9324_X401".DigitalInput08; (*Bag arrived CDC5 (Line 8)*)
	OK[14] AT %IX."X20DM9324_X409".ModuleOk;
	X[4].X09 AT %IX."X20DM9324_X409".DigitalInput01; (*Bag arrived CP2 buffer*)
	X[4].X10 AT %IX."X20DM9324_X409".DigitalInput02; (*CP2 Bag at buffer stop*)
	X[4].X11 AT %IX."X20DM9324_X409".DigitalInput03; (*CIC1 Bag at buffer *)
	X[4].X12 AT %IX."X20DM9324_X409".DigitalInput04; (*CIC2 Bag at buffer*)
	X[4].X13 AT %IX."X20DM9324_X409".DigitalInput05; (*CDC 2 Full bag buffer*)
	X[4].X14 AT %IX."X20DM9324_X409".DigitalInput06; (*CP3 Bag at buffer*)
	X[4].X15 AT %IX."X20DM9324_X409".DigitalInput07; (*CDC 1 Full bag buffer*)
	X[4].X16 AT %IX."X20DM9324_X409".DigitalInput08; (*CSR 3 Bag at buffer*)
	OK[15] AT %IX."X20DO8332_Y401".ModuleOk;
	Y[4].Y01 AT %QX."X20DO8332_Y401".DigitalOutput01; (*Ongoing select line 1*)
	Y[4].Y02 AT %QX."X20DO8332_Y401".DigitalOutput02; (*Ongoing select line 2*)
	Y[4].Y03 AT %QX."X20DO8332_Y401".DigitalOutput03; (*Ongoing select line 3*)
	Y[4].Y04 AT %QX."X20DO8332_Y401".DigitalOutput04; (*Ongoing select line 4*)
	Y[4].Y05 AT %QX."X20DO8332_Y401".DigitalOutput05; (*Ongoing select line 5*)
	Y[4].Y06 AT %QX."X20DO8332_Y401".DigitalOutput06; (*Ongoing select line 6*)
	Y[4].Y07 AT %QX."X20DO8332_Y401".DigitalOutput07; (*CP2 line 7*)
	Y[4].Y08 AT %QX."X20DO8332_Y401".DigitalOutput08; (*CP2 line 8*)
	OK[16] AT %IX."X20DO8332_Y409".ModuleOk;
	Y[4].Y09 AT %QX."X20DO8332_Y409".DigitalOutput01; (*Ongoing reset lines*)
	Y[4].Y10 AT %QX."X20DO8332_Y409".DigitalOutput02; (*CP 3 Stop and point*)
	Y[4].Y11 AT %QX."X20DO8332_Y409".DigitalOutput03; (*CP 3 Stop and point*)
	Y[4].Y12 AT %QX."X20DO8332_Y409".DigitalOutput04; (*CP 2 Buffer stop*)
	Y[4].Y13 AT %QX."X20DO8332_Y409".DigitalOutput05; (*CIC 1 Buffer stop*)
	Y[4].Y14 AT %QX."X20DO8332_Y409".DigitalOutput06; (*CIC 2 Buffer stop*)
	Y[4].Y15 AT %QX."X20DO8332_Y409".DigitalOutput07; (*CIC 3 Buffer stop*)
	Y[4].Y16 AT %QX."X20DO8332_Y409".DigitalOutput08; (*CIC 4 Buffer stop*)
	OK[17] AT %IX."X20DM9324_X501".ModuleOk;
	X[5].X01 AT %IX."X20DM9324_X501".DigitalInput01; (*Offgoing bag at line 1 stop*)
	X[5].X02 AT %IX."X20DM9324_X501".DigitalInput02; (*Offgoing bag at line 2 stop*)
	X[5].X03 AT %IX."X20DM9324_X501".DigitalInput03; (*Offgoing bag at line 3 stop*)
	X[5].X04 AT %IX."X20DM9324_X501".DigitalInput04; (*Offgoing bag at line 4 stop*)
	X[5].X05 AT %IX."X20DM9324_X501".DigitalInput05; (*Offgoing bag at line 5 stop*)
	X[5].X06 AT %IX."X20DM9324_X501".DigitalInput06; (*Offgoing bag at line 6 stop*)
	X[5].X07 AT %IX."X20DM9324_X501".DigitalInput07; (*CVC 1 bag on carriage*)
	X[5].X08 AT %IX."X20DM9324_X501".DigitalInput08; (*CIC1 Bag at buffer stop*)
	OK[18] AT %IX."X20DM9324_X509".ModuleOk;
	X[5].X09 AT %IX."X20DM9324_X509".DigitalInput01; (*CIC1 Paddle *)
	X[5].X10 AT %IX."X20DM9324_X509".DigitalInput02; (*CIC 1 Bag at bottom*)
	X[5].X11 AT %IX."X20DM9324_X509".DigitalInput03; (*CIC2 Bag at buffer stop*)
	X[5].X12 AT %IX."X20DM9324_X509".DigitalInput04; (*CIC2 Paddle*)
	X[5].X13 AT %IX."X20DM9324_X509".DigitalInput05; (*CIC2 Bag at bottom*)
	X[5].X14 AT %IX."X20DM9324_X509".DigitalInput06; (*Bag at CDC1 empty buffer stop*)
	X[5].X15 AT %IX."X20DM9324_X509".DigitalInput07; (*Bag at CDC2 empty buffer stop*)
	X[5].X16 AT %IX."X20DM9324_X509".DigitalInput08; (*CP 6 Bag at buffer*)
	OK[19] AT %IX."X20DO8332_Y501".ModuleOk;
	Y[5].Y01 AT %QX."X20DO8332_Y501".DigitalOutput01; (*Offgoing select line 1*)
	Y[5].Y02 AT %QX."X20DO8332_Y501".DigitalOutput02; (*Offgoing select line 2*)
	Y[5].Y03 AT %QX."X20DO8332_Y501".DigitalOutput03; (*Offgoing select line 3*)
	Y[5].Y04 AT %QX."X20DO8332_Y501".DigitalOutput04; (*Offgoing select line 4*)
	Y[5].Y05 AT %QX."X20DO8332_Y501".DigitalOutput05; (*Offgoing select line 5*)
	Y[5].Y06 AT %QX."X20DO8332_Y501".DigitalOutput06; (*Offgoing select line 6*)
	Y[5].Y07 AT %QX."X20DO8332_Y501".DigitalOutput07; (*Offgoing reset*)
	Y[5].Y08 AT %QX."X20DO8332_Y501".DigitalOutput08; (*CDC 1 Select CP5*)
	OK[20] AT %IX."X20DO8332_Y509".ModuleOk;
	Y[5].Y09 AT %QX."X20DO8332_Y509".DigitalOutput01; (*CDC 2 Select CP4*)
	Y[5].Y10 AT %QX."X20DO8332_Y509".DigitalOutput02; (*CDC3 Select CP4 and CP5*)
	Y[5].Y11 AT %QX."X20DO8332_Y509".DigitalOutput03; (*CPC 1 Low level buffer stop*)
	Y[5].Y12 AT %QX."X20DO8332_Y509".DigitalOutput04; (*CDC 1 Empty bag buffer stop and point*)
	Y[5].Y13 AT %QX."X20DO8332_Y509".DigitalOutput05; (*CDC 2 Empty bag buffer stop and point*)
	Y[5].Y14 AT %QX."X20DO8332_Y509".DigitalOutput06; (*CSR 1 Speed reducor 1*)
	Y[5].Y15 AT %QX."X20DO8332_Y509".DigitalOutput07; (*CSR 2 Speed reducor 2*)
	Y[5].Y16 AT %QX."X20DO8332_Y509".DigitalOutput08; (*CPR 1 Pressure releif 1 stop*)
	OK[21] AT %IX."X20DM9324_X601".ModuleOk;
	X[6].X01 AT %IX."X20DM9324_X601".DigitalInput01; (*CPC 1 Bag at low level buffer stop*)
	X[6].X02 AT %IX."X20DM9324_X601".DigitalInput02; (*CPC1 Carriage at bottom*)
	X[6].X03 AT %IX."X20DM9324_X601".DigitalInput03; (*CPC1 Carriage at top*)
	X[6].X04 AT %IX."X20DM9324_X601".DigitalInput04; (*CPC1 Bag out at top*)
	X[6].X05 AT %IX."X20DM9324_X601".DigitalInput05; (*CDC1 Bag at buffer stop*)
	X[6].X06 AT %IX."X20DM9324_X601".DigitalInput06; (*CDC1 Bag in discharger*)
	X[6].X07 AT %IX."X20DM9324_X601".DigitalInput07; (*CDC1 Bag out of discharger*)
	X[6].X08 AT %IX."X20DM9324_X601".DigitalInput08; (*CDC1 Drop load (Test)*)
	OK[22] AT %IX."X20DM9324_X609".ModuleOk;
	X[6].X09 AT %IX."X20DM9324_X609".DigitalInput01; (*CDC2 Bag at buffer stop*)
	X[6].X10 AT %IX."X20DM9324_X609".DigitalInput02; (*CDC2 Bag in discharger*)
	X[6].X11 AT %IX."X20DM9324_X609".DigitalInput03; (*CDC2 Bag out of discharger*)
	X[6].X12 AT %IX."X20DM9324_X609".DigitalInput04; (*CDC2 Drop load (Test)*)
	X[6].X13 AT %IX."X20DM9324_X609".DigitalInput05; (*CDC3 Bag at buffer stop*)
	X[6].X14 AT %IX."X20DM9324_X609".DigitalInput06; (*CDC3 Bag in discharger*)
	X[6].X15 AT %IX."X20DM9324_X609".DigitalInput07; (*CIC 3 Bag at buffer*)
	X[6].X16 AT %IX."X20DM9324_X609".DigitalInput08; (*CDC3 Drop load (Test)*)
	OK[23] AT %IX."X20DO8332_Y601".ModuleOk;
	Y[6].Y01 AT %QX."X20DO8332_Y601".DigitalOutput01; (*CDC1 Buffer stop*)
	Y[6].Y02 AT %QX."X20DO8332_Y601".DigitalOutput02; (*CDC1 Steady cylinders*)
	Y[6].Y03 AT %QX."X20DO8332_Y601".DigitalOutput03; (*CDC1 Open bag*)
	Y[6].Y04 AT %QX."X20DO8332_Y601".DigitalOutput04; (*CDC1 Close bag*)
	Y[6].Y05 AT %QX."X20DO8332_Y601".DigitalOutput05; (*CDC1 Discharger stop*)
	Y[6].Y06 AT %QX."X20DO8332_Y601".DigitalOutput06; (*CDC1 Bag ready*)
	Y[6].Y07 AT %QX."X20DO8332_Y601".DigitalOutput07; (*CDC2 Buffer stop*)
	Y[6].Y08 AT %QX."X20DO8332_Y601".DigitalOutput08; (*CDC2 Steady cylinders*)
	OK[24] AT %IX."X20DO8332_Y609".ModuleOk;
	Y[6].Y09 AT %QX."X20DO8332_Y609".DigitalOutput01; (*CDC2 Open bag*)
	Y[6].Y10 AT %QX."X20DO8332_Y609".DigitalOutput02; (*CDC2 Close bag*)
	Y[6].Y11 AT %QX."X20DO8332_Y609".DigitalOutput03; (*CDC2 Discharger stop*)
	Y[6].Y12 AT %QX."X20DO8332_Y609".DigitalOutput04; (*CDC2 Bag ready*)
	Y[6].Y13 AT %QX."X20DO8332_Y609".DigitalOutput05; (*CDC3 Buffer stop*)
	Y[6].Y14 AT %QX."X20DO8332_Y609".DigitalOutput06; (*CDC3 Steady cylinders*)
	Y[6].Y15 AT %QX."X20DO8332_Y609".DigitalOutput07; (*CDC3 Open bag*)
	Y[6].Y16 AT %QX."X20DO8332_Y609".DigitalOutput08; (*CDC3 Close bag*)
	OK[25] AT %IX."X20DM9324_X701".ModuleOk;
	X[7].X01 AT %IX."X20DM9324_X701".DigitalInput01; (*CDC4 Bag at buffer stop*)
	X[7].X02 AT %IX."X20DM9324_X701".DigitalInput02; (*CDC4 Bag in discharger*)
	X[7].X03 AT %IX."X20DM9324_X701".DigitalInput03; (*CDC4 Bag out of discharger*)
	X[7].X04 AT %IX."X20DM9324_X701".DigitalInput04; (*CDC4 Drop load*)
	X[7].X05 AT %IX."X20DM9324_X701".DigitalInput05; (*CBC1 Bag at buffer stop*)
	X[7].X06 AT %IX."X20DM9324_X701".DigitalInput06; (*CBC1 Bag in discharger*)
	X[7].X07 AT %IX."X20DM9324_X701".DigitalInput07; (*CBC1 Bag out of discharger*)
	X[7].X08 AT %IX."X20DM9324_X701".DigitalInput08; (*Spare*)
	OK[26] AT %IX."X20DM9324_X709".ModuleOk;
	X[7].X09 AT %IX."X20DM9324_X709".DigitalInput01; (*CPI1 Bag at buffer stop*)
	X[7].X10 AT %IX."X20DM9324_X709".DigitalInput02; (*CPI1 Bag at bottom*)
	X[7].X11 AT %IX."X20DM9324_X709".DigitalInput03; (*CPI1 Carriage at top*)
	X[7].X12 AT %IX."X20DM9324_X709".DigitalInput04; (*CPI1 Carriage at bottom*)
	X[7].X13 AT %IX."X20DM9324_X709".DigitalInput05; (*CPI1 Bag out at top*)
	X[7].X14 AT %IX."X20DM9324_X709".DigitalInput06; (*CPI2 Bag at buffer stop*)
	X[7].X15 AT %IX."X20DM9324_X709".DigitalInput07; (*CPI2 Bag at bottom*)
	X[7].X16 AT %IX."X20DM9324_X709".DigitalInput08; (*CPI2 Carriage at top*)
	OK[27] AT %IX."X20DO8332_Y701".ModuleOk;
	Y[7].Y01 AT %QX."X20DO8332_Y701".DigitalOutput01; (*CDC3 Discharger stop*)
	Y[7].Y02 AT %QX."X20DO8332_Y701".DigitalOutput02; (*CDC3 Bag ready*)
	Y[7].Y03 AT %QX."X20DO8332_Y701".DigitalOutput03; (*CDC4 Bag at buffer stop*)
	Y[7].Y04 AT %QX."X20DO8332_Y701".DigitalOutput04; (*CDC4 Steady cylinders*)
	Y[7].Y05 AT %QX."X20DO8332_Y701".DigitalOutput05; (*CDC4 Open bag*)
	Y[7].Y06 AT %QX."X20DO8332_Y701".DigitalOutput06; (*CDC4 Close bag*)
	Y[7].Y07 AT %QX."X20DO8332_Y701".DigitalOutput07; (*CDC4 Discharger stop*)
	Y[7].Y08 AT %QX."X20DO8332_Y701".DigitalOutput08; (*CDC4 Bag ready*)
	OK[28] AT %IX."X20DO8332_Y709".ModuleOk;
	Y[7].Y09 AT %QX."X20DO8332_Y709".DigitalOutput01; (*CBC1 Open buffer stop*)
	Y[7].Y10 AT %QX."X20DO8332_Y709".DigitalOutput02; (*CBC1 Steady cylinders*)
	Y[7].Y11 AT %QX."X20DO8332_Y709".DigitalOutput03; (*CBC1 Open bag*)
	Y[7].Y12 AT %QX."X20DO8332_Y709".DigitalOutput04; (*CBC1 Close bag*)
	Y[7].Y13 AT %QX."X20DO8332_Y709".DigitalOutput05; (*CBC1 Discharger stop*)
	Y[7].Y14 AT %QX."X20DO8332_Y709".DigitalOutput06; (*Spare*)
	Y[7].Y15 AT %QX."X20DO8332_Y709".DigitalOutput07; (*Spare*)
	Y[7].Y16 AT %QX."X20DO8332_Y709".DigitalOutput08; (*Spare*)
	OK[29] AT %IX."X20DM9324_X801".ModuleOk;
	X[8].X01 AT %IX."X20DM9324_X801".DigitalInput01; (*CPI2 Carriage at bottom*)
	X[8].X02 AT %IX."X20DM9324_X801".DigitalInput02; (*CPI2 Bag out at top*)
	X[8].X03 AT %IX."X20DM9324_X801".DigitalInput03; (*CPI3 Bag at buffer stop*)
	X[8].X04 AT %IX."X20DM9324_X801".DigitalInput04; (*CPI3 Bag at bottom*)
	X[8].X05 AT %IX."X20DM9324_X801".DigitalInput05; (*CPI3 Carriage at top*)
	X[8].X06 AT %IX."X20DM9324_X801".DigitalInput06; (*CPI3 Carriage at bottom*)
	X[8].X07 AT %IX."X20DM9324_X801".DigitalInput07; (*CPI3 Bag out at top*)
	X[8].X08 AT %IX."X20DM9324_X801".DigitalInput08; (*CIC 3 Bag at buffer stop*)
	OK[30] AT %IX."X20DM9324_X809".ModuleOk;
	X[8].X09 AT %IX."X20DM9324_X809".DigitalInput01; (*CIC3 Paddle in position*)
	X[8].X10 AT %IX."X20DM9324_X809".DigitalInput02; (*CIC3 Bag at bottom*)
	X[8].X11 AT %IX."X20DM9324_X809".DigitalInput03; (*CIC3 Bag out at top*)
	X[8].X12 AT %IX."X20DM9324_X809".DigitalInput04; (*Spare*)
	X[8].X13 AT %IX."X20DM9324_X809".DigitalInput05; (*CIC 4 Bag at buffer*)
	X[8].X14 AT %IX."X20DM9324_X809".DigitalInput06; (*CLU 1 bag at empty buffer*)
	X[8].X15 AT %IX."X20DM9324_X809".DigitalInput07; (*CLU 2 bag at empty buffer*)
	X[8].X16 AT %IX."X20DM9324_X809".DigitalInput08; (*Bag at CP 9 buffer stop*)
	OK[31] AT %IX."X20DO8332_Y801".ModuleOk;
	Y[8].Y01 AT %QX."X20DO8332_Y801".DigitalOutput01; (*CDC4 Alarm (new 2\5\04)*)
	Y[8].Y02 AT %QX."X20DO8332_Y801".DigitalOutput02; (*CDC5 Alarm (new 2\5\04)*)
	Y[8].Y03 AT %QX."X20DO8332_Y801".DigitalOutput03; (*CP7  empty buffer stop after CP 6*)
	Y[8].Y04 AT %QX."X20DO8332_Y801".DigitalOutput04; (*CP7 empty buffer stop after CPI4*)
	Y[8].Y05 AT %QX."X20DO8332_Y801".DigitalOutput05; (*CP9 To CLU1 empty bag buffer*)
	Y[8].Y06 AT %QX."X20DO8332_Y801".DigitalOutput06; (*CP9 To CLU2 empty bag buffer*)
	Y[8].Y07 AT %QX."X20DO8332_Y801".DigitalOutput07; (*CP9 Buffer stop*)
	Y[8].Y08 AT %QX."X20DO8332_Y801".DigitalOutput08; (*Select CP 8 to CP 7*)
	OK[32] AT %IX."X20DO8332_Y809".ModuleOk;
	Y[8].Y09 AT %QX."X20DO8332_Y809".DigitalOutput01; (*Select CP 8 to CDC 3*)
	Y[8].Y10 AT %QX."X20DO8332_Y809".DigitalOutput02; (*Spare*)
	Y[8].Y11 AT %QX."X20DO8332_Y809".DigitalOutput03; (*Spare*)
	Y[8].Y12 AT %QX."X20DO8332_Y809".DigitalOutput04; (*Spare*)
	Y[8].Y13 AT %QX."X20DO8332_Y809".DigitalOutput05; (*CIC 5 Run incline*)
	Y[8].Y14 AT %QX."X20DO8332_Y809".DigitalOutput06; (*CIC 6 Run incline*)
	Y[8].Y15 AT %QX."X20DO8332_Y809".DigitalOutput07; (*CP 15 Move carriage down*)
	Y[8].Y16 AT %QX."X20DO8332_Y809".DigitalOutput08; (*CP 16 Move carriage down*)
	OK[33] AT %IX."X20DM9324_X901".ModuleOk;
	X[9].X01 AT %IX."X20DM9324_X901".DigitalInput01; (*CPC 1 Bag at buffer*)
	X[9].X02 AT %IX."X20DM9324_X901".DigitalInput02; (*CPC 1 Bag on carriage*)
	X[9].X03 AT %IX."X20DM9324_X901".DigitalInput03; (*CPR 1 Bag at stop*)
	X[9].X04 AT %IX."X20DM9324_X901".DigitalInput04; (*CPR 1 Line full*)
	X[9].X05 AT %IX."X20DM9324_X901".DigitalInput05; (*FVC 1 Up push button*)
	X[9].X06 AT %IX."X20DM9324_X901".DigitalInput06; (*CDC 3 Bag at buffer*)
	X[9].X07 AT %IX."X20DM9324_X901".DigitalInput07; (*CDC 4 Bag at buffer*)
	X[9].X08 AT %IX."X20DM9324_X901".DigitalInput08; (*CPR 2 Bag at buffer stop*)
	OK[34] AT %IX."X20DM9324_X909".ModuleOk;
	X[9].X09 AT %IX."X20DM9324_X909".DigitalInput01; (*CIC 4 Paddle in position*)
	X[9].X10 AT %IX."X20DM9324_X909".DigitalInput02; (*CIC 4 Bag at buffer stop*)
	X[9].X11 AT %IX."X20DM9324_X909".DigitalInput03; (*CIC 4 Bag at bottom*)
	X[9].X12 AT %IX."X20DM9324_X909".DigitalInput04; (*CPR 3 Bag at buffer stop*)
	X[9].X13 AT %IX."X20DM9324_X909".DigitalInput05; (*CPR 3 Line full*)
	X[9].X14 AT %IX."X20DM9324_X909".DigitalInput06; (*CP 3 Bag at buffer stop*)
	X[9].X15 AT %IX."X20DM9324_X909".DigitalInput07; (*CPI 4 Bag at buffer stop*)
	X[9].X16 AT %IX."X20DM9324_X909".DigitalInput08; (*CPI 4 Bag at bottom*)
	OK[35] AT %IX."X20DO8332_Y901".ModuleOk;
	Y[9].Y01 AT %QX."X20DO8332_Y901".DigitalOutput01; (*Spare*)
	Y[9].Y02 AT %QX."X20DO8332_Y901".DigitalOutput02; (*Spare*)
	Y[9].Y03 AT %QX."X20DO8332_Y901".DigitalOutput03; (*Spare*)
	Y[9].Y04 AT %QX."X20DO8332_Y901".DigitalOutput04; (*Spare*)
	Y[9].Y05 AT %QX."X20DO8332_Y901".DigitalOutput05; (*CSR 2 Close speed reducor *)
	Y[9].Y06 AT %QX."X20DO8332_Y901".DigitalOutput06; (*Spare*)
	Y[9].Y07 AT %QX."X20DO8332_Y901".DigitalOutput07; (*Spare*)
	Y[9].Y08 AT %QX."X20DO8332_Y901".DigitalOutput08; (*CPR 2 Open buffer stop *)
	OK[36] AT %IX."X20DO8332_Y909".ModuleOk;
	Y[9].Y09 AT %QX."X20DO8332_Y909".DigitalOutput01; (*Spare*)
	Y[9].Y10 AT %QX."X20DO8332_Y909".DigitalOutput02; (*Spare*)
	Y[9].Y11 AT %QX."X20DO8332_Y909".DigitalOutput03; (*Spare*)
	Y[9].Y12 AT %QX."X20DO8332_Y909".DigitalOutput04; (*CPR 3 Open buffer stop*)
	Y[9].Y13 AT %QX."X20DO8332_Y909".DigitalOutput05; (*Spare*)
	Y[9].Y14 AT %QX."X20DO8332_Y909".DigitalOutput06; (*Spare*)
	Y[9].Y15 AT %QX."X20DO8332_Y909".DigitalOutput07; (*Spare*)
	Y[9].Y16 AT %QX."X20DO8332_Y909".DigitalOutput08; (*Spare*)
	OK[37] AT %IX."X20DM9324_X1001".ModuleOk;
	X[10].X01 AT %IX."X20DM9324_X1001".DigitalInput01; (*CPI 4 Carriage at bottom*)
	X[10].X02 AT %IX."X20DM9324_X1001".DigitalInput02; (*CPI 4 Carriage at top*)
	X[10].X03 AT %IX."X20DM9324_X1001".DigitalInput03; (*CPI 4 Bag out at top*)
	X[10].X04 AT %IX."X20DM9324_X1001".DigitalInput04; (*CP 7 Bag at buffer stop *)
	X[10].X05 AT %IX."X20DM9324_X1001".DigitalInput05; (*CP 7 Bag at buffer stop*)
	X[10].X06 AT %IX."X20DM9324_X1001".DigitalInput06; (*CPI 2 Bag at buffer    *)
	X[10].X07 AT %IX."X20DM9324_X1001".DigitalInput07; (*CIC 5 Bag at bottom*)
	X[10].X08 AT %IX."X20DM9324_X1001".DigitalInput08; (*CIC 5 Paddle in position*)
	OK[38] AT %IX."X20DM9324_X1009".ModuleOk;
	X[10].X09 AT %IX."X20DM9324_X1009".DigitalInput01; (*CIC 5 Bag at buffer stop*)
	X[10].X10 AT %IX."X20DM9324_X1009".DigitalInput02; (*CIC 5 Bag at buffer*)
	X[10].X11 AT %IX."X20DM9324_X1009".DigitalInput03; (*CIC 6 Bag at buffer*)
	X[10].X12 AT %IX."X20DM9324_X1009".DigitalInput04; (*CIC 6 Bag at bottom*)
	X[10].X13 AT %IX."X20DM9324_X1009".DigitalInput05; (*CIC 6 Paddle in position*)
	X[10].X14 AT %IX."X20DM9324_X1009".DigitalInput06; (*CP 14 Bag at buffer stop*)
	X[10].X15 AT %IX."X20DM9324_X1009".DigitalInput07; (*CBC 1 Bag at buffer*)
	X[10].X16 AT %IX."X20DM9324_X1009".DigitalInput08; (*CPR 2 Line full*)
	OK[39] AT %IX."X20DO8332_Y1001".ModuleOk;
	Y[10].Y01 AT %QX."X20DO8332_Y1001".DigitalOutput01; (*CP 10 Select point to CP11*)
	Y[10].Y02 AT %QX."X20DO8332_Y1001".DigitalOutput02; (*CP 11 Select point to CIC 5*)
	Y[10].Y03 AT %QX."X20DO8332_Y1001".DigitalOutput03; (*CP 12 Select point to CP 13*)
	Y[10].Y04 AT %QX."X20DO8332_Y1001".DigitalOutput04; (*CP 13 Select point to CIC 6*)
	Y[10].Y05 AT %QX."X20DO8332_Y1001".DigitalOutput05; (*Spare*)
	Y[10].Y06 AT %QX."X20DO8332_Y1001".DigitalOutput06; (*Spare*)
	Y[10].Y07 AT %QX."X20DO8332_Y1001".DigitalOutput07; (*Spare*)
	Y[10].Y08 AT %QX."X20DO8332_Y1001".DigitalOutput08; (*Spare*)
	OK[40] AT %IX."X20DO8332_Y1009".ModuleOk;
	Y[10].Y09 AT %QX."X20DO8332_Y1009".DigitalOutput01; (*Spare*)
	Y[10].Y10 AT %QX."X20DO8332_Y1009".DigitalOutput02; (*CPR 4 Open stop*)
	Y[10].Y11 AT %QX."X20DO8332_Y1009".DigitalOutput03; (*Spare*)
	Y[10].Y12 AT %QX."X20DO8332_Y1009".DigitalOutput04; (*Spare*)
	Y[10].Y13 AT %QX."X20DO8332_Y1009".DigitalOutput05; (*CP 17 Select point from CP16*)
	Y[10].Y14 AT %QX."X20DO8332_Y1009".DigitalOutput06; (*CP 14 Select buffer stop and point*)
	Y[10].Y15 AT %QX."X20DO8332_Y1009".DigitalOutput07; (*CP 15 Select point from CPI5*)
	Y[10].Y16 AT %QX."X20DO8332_Y1009".DigitalOutput08; (*CP 16 Select point from CP15*)
	OK[47] AT %IX."X20DM9324_X1101".ModuleOk;
	X[11].X01 AT %IX."X20DM9324_X1101".DigitalInput01; (*CP I5 Carriage at top *)
	X[11].X02 AT %IX."X20DM9324_X1101".DigitalInput02; (*CP I5 Carriage at bottom *)
	X[11].X03 AT %IX."X20DM9324_X1101".DigitalInput03; (*CP I5 Bag at bottom *)
	X[11].X04 AT %IX."X20DM9324_X1101".DigitalInput04; (*CP16 Bag at buffer *)
	X[11].X05 AT %IX."X20DM9324_X1101".DigitalInput05; (*CP16 Bag at buffer stop *)
	X[11].X06 AT %IX."X20DM9324_X1101".DigitalInput06; (*CP I6 Carriage at top  *)
	X[11].X07 AT %IX."X20DM9324_X1101".DigitalInput07; (*CP I6 Carriage at bottom *)
	X[11].X08 AT %IX."X20DM9324_X1101".DigitalInput08; (*CPI 6 Bag at bottom*)
	OK[48] AT %IX."X20DM9324_X1109".ModuleOk;
	X[11].X09 AT %IX."X20DM9324_X1109".DigitalInput01; (*CPR 4 Line full *)
	X[11].X10 AT %IX."X20DM9324_X1109".DigitalInput02; (*CPR 4 Bag at stop *)
	X[11].X11 AT %IX."X20DM9324_X1109".DigitalInput03; (*Spare*)
	X[11].X12 AT %IX."X20DM9324_X1109".DigitalInput04; (*Spare*)
	X[11].X13 AT %IX."X20DM9324_X1109".DigitalInput05; (*Spare*)
	X[11].X14 AT %IX."X20DM9324_X1109".DigitalInput06; (*Spare*)
	X[11].X15 AT %IX."X20DM9324_X1109".DigitalInput07; (*Spare*)
	X[11].X16 AT %IX."X20DM9324_X1109".DigitalInput08; (*Spare*)
	OK[49] AT %IX."X20DO8332_Y1101".ModuleOk;
	Y[11].Y01 AT %QX."X20DO8332_Y1101".DigitalOutput01; (*CVC1 Carriage up*)
	Y[11].Y02 AT %QX."X20DO8332_Y1101".DigitalOutput02; (*CVC1 Carriage down*)
	Y[11].Y03 AT %QX."X20DO8332_Y1101".DigitalOutput03; (*CVC1 Carriage stop*)
	Y[11].Y04 AT %QX."X20DO8332_Y1101".DigitalOutput04; (*CIC1 Run motor*)
	Y[11].Y05 AT %QX."X20DO8332_Y1101".DigitalOutput05; (*CIC2 Run motor*)
	Y[11].Y06 AT %QX."X20DO8332_Y1101".DigitalOutput06; (*CIC3 Run motor*)
	Y[11].Y07 AT %QX."X20DO8332_Y1101".DigitalOutput07; (*CPI1 Carriage down*)
	Y[11].Y08 AT %QX."X20DO8332_Y1101".DigitalOutput08; (*CPI2 Carriage down*)
	OK[50] AT %IX."X20DO8332_Y1109".ModuleOk;
	Y[11].Y09 AT %QX."X20DO8332_Y1109".DigitalOutput01; (*CPI3 Carriage down*)
	Y[11].Y10 AT %QX."X20DO8332_Y1109".DigitalOutput02; (*CPC1 Carriage up*)
	Y[11].Y11 AT %QX."X20DO8332_Y1109".DigitalOutput03; (*CPC1 Carriage down*)
	Y[11].Y12 AT %QX."X20DO8332_Y1109".DigitalOutput04; (*CPC1 Carriage stop*)
	Y[11].Y13 AT %QX."X20DO8332_Y1109".DigitalOutput05; (*Run Belt A*)
	Y[11].Y14 AT %QX."X20DO8332_Y1109".DigitalOutput06; (*Run Belt B*)
	Y[11].Y15 AT %QX."X20DO8332_Y1109".DigitalOutput07; (*CIC4 Run motor*)
	Y[11].Y16 AT %QX."X20DO8332_Y1109".DigitalOutput08; (*CPI6 Carriage down*)
	StnOK[1] AT %IX."X20AI4222_SS1_4".ModuleOk;
	::AI1223[1] AT %IW."X20AI4222_SS1_4".AnalogInput01;
	::AI1223[2] AT %IW."X20AI4222_SS1_4".AnalogInput02;
	::AI1223[3] AT %IW."X20AI4222_SS1_4".AnalogInput03;
	::AI1223[4] AT %IW."X20AI4222_SS1_4".AnalogInput04;
	::AI1223[5] AT %IW."X20AI4222_SS5_8".AnalogInput01;
	::AI1223[6] AT %IW."X20AI4222_SS5_8".AnalogInput02;
	::AI1223[7] AT %IW."X20AI4222_SS5_8".AnalogInput03;
	::AI1223[8] AT %IW."X20AI4222_SS5_8".AnalogInput04;
	::AI1223[9] AT %IW."X20AI4222_SS9_12".AnalogInput01;
	::AI1223[10] AT %IW."X20AI4222_SS9_12".AnalogInput02;
	::AI1223[11] AT %IW."X20AI4222_SS9_12".AnalogInput03;
	::AI1223[12] AT %IW."X20AI4222_SS9_12".AnalogInput04;
	::AI1223[13] AT %IW."X20AI4222_SS13_14".AnalogInput01;
	::AI1223[14] AT %IW."X20AI4222_SS13_14".AnalogInput02;
	Y[12].Y01 AT %QX."X20DO8332_Y12".DigitalOutput01; (*SS 1 Lamp*)
	Y[12].Y02 AT %QX."X20DO8332_Y12".DigitalOutput02; (*SS 2 Lamp*)
	Y[12].Y03 AT %QX."X20DO8332_Y12".DigitalOutput03; (*SS 3 Lamp*)
	Y[12].Y04 AT %QX."X20DO8332_Y12".DigitalOutput04; (*SS 4 Lamp*)
	Y[12].Y05 AT %QX."X20DO8332_Y12".DigitalOutput05; (*SS 1 Open Bag*)
	Y[12].Y06 AT %QX."X20DO8332_Y12".DigitalOutput06; (*SS 2 Open Bag*)
	Y[12].Y07 AT %QX."X20DO8332_Y12".DigitalOutput07; (*SS 3 Open Bag*)
	Y[12].Y08 AT %QX."X20DO8332_Y12".DigitalOutput08; (*SS 4 Open Bag*)
	Y[13].Y01 AT %QX."X20DO8332_Y13".DigitalOutput01; (*SS 5 Lamp*)
	::Y[13].Y02 AT %QX."X20DO8332_Y13".DigitalOutput02; (*SS 6 Lamp*)
	::Y[13].Y03 AT %QX."X20DO8332_Y13".DigitalOutput03; (*SS 7 Lamp*)
	::Y[13].Y04 AT %QX."X20DO8332_Y13".DigitalOutput04; (*Spare*)
	::Y[13].Y05 AT %QX."X20DO8332_Y13".DigitalOutput05; (*SS 5 Open Bag*)
	::Y[13].Y06 AT %QX."X20DO8332_Y13".DigitalOutput06; (*SS 6 Open Bag*)
	::Y[13].Y07 AT %QX."X20DO8332_Y13".DigitalOutput07; (*SS 7 Open Bag*)
	::Y[13].Y08 AT %QX."X20DO8332_Y13".DigitalOutput08; (*Spare*)
	::Y[14].Y01 AT %QX."X20DO8332_Y14".DigitalOutput01; (*SS 8 Lamp*)
	Y[14].Y02 AT %QX."X20DO8332_Y14".DigitalOutput02; (*SS 9 Lamp*)
	Y[14].Y03 AT %QX."X20DO8332_Y14".DigitalOutput03; (*SS 10 Lamp*)
	Y[14].Y04 AT %QX."X20DO8332_Y14".DigitalOutput04; (*SS 11 Lamp*)
	Y[14].Y05 AT %QX."X20DO8332_Y14".DigitalOutput05; (*SS 8 Open Bag*)
	Y[14].Y06 AT %QX."X20DO8332_Y14".DigitalOutput06; (*SS 9 Open Bag*)
	Y[14].Y07 AT %QX."X20DO8332_Y14".DigitalOutput07; (*SS 10 Open Bag*)
	Y[14].Y08 AT %QX."X20DO8332_Y14".DigitalOutput08; (*SS 11 Open Bag*)
	Y[15].Y01 AT %QX."X20DO8332_Y15".DigitalOutput01; (*SS 12 Lamp*)
	Y[15].Y02 AT %QX."X20DO8332_Y15".DigitalOutput02; (*SS 13 Lamp*)
	Y[15].Y03 AT %QX."X20DO8332_Y15".DigitalOutput03; (*SS 14 Lamp*)
	Y[15].Y04 AT %QX."X20DO8332_Y15".DigitalOutput04; (*Spare*)
	Y[15].Y05 AT %QX."X20DO8332_Y15".DigitalOutput05; (*SS 12 Open Bag*)
	Y[15].Y06 AT %QX."X20DO8332_Y15".DigitalOutput06; (*SS 13 Open Bag*)
	Y[15].Y07 AT %QX."X20DO8332_Y15".DigitalOutput07; (*SS 14 Open Bag*)
	Y[15].Y08 AT %QX."X20DO8332_Y15".DigitalOutput08; (*Spare*)
	X[15].X01 AT %IX."X20DM9324_X15".DigitalInput01; (*Spare*)
	X[15].X02 AT %IX."X20DM9324_X15".DigitalInput02; (*Spare*)
	X[15].X03 AT %IX."X20DM9324_X15".DigitalInput03; (*Spare*)
	X[15].X04 AT %IX."X20DM9324_X15".DigitalInput04; (*Belt 1 key switch*)
	X[15].X05 AT %IX."X20DM9324_X15".DigitalInput05; (*Spare*)
	X[15].X06 AT %IX."X20DM9324_X15".DigitalInput06; (*Spare*)
	X[15].X07 AT %IX."X20DM9324_X15".DigitalInput07; (*Spare*)
	X[15].X08 AT %IX."X20DM9324_X15".DigitalInput08; (*Belt 2 key switch*)
END_VAR
```

- Safety project (password-protected, skipped)

## Logical view

Binary libraries used (declarations not repeated): standard, runtime, FileIO, Ethernet, dvframe, DataObj, OPERATOR, AsTime, AsString, AsCANopen, SupLib4, sys_lib, AsTCP, KGstring, CAN_Lib, Visapi, AsARCfg, AsETH, AsDb, brsystem, AsUSB, WETCAN2, AsMem, AsArLog, AsBrWStr, AsUDP, AsIODiag, AsBrStr, AsIecCon, IecCheck, AsXml, AsPciStr, AsIOAcc, AsBrMath, MpServer, AsHttp, SUP 1.00.0, AsSafety, MTTypes 1.03.0, MTBasics 2.21.0, AsEPL

### Package Logical/GlobalVariables - Global Variables

### Package Logical/GlobalVariables/Alarm - Alarm Variables

### Alarm.var
```iecst
VAR
	SpecialTreatment : ARRAY[0..9] OF UINT;
	LoadingBagLU1 : BOOL;
	StrobeComplete4 : BOOL;
	StrobeComplete3 : BOOL;
	StrobeComplete2 : BOOL;
	StrobeComplete1 : BOOL;
	Alarm : ARRAY[0..209] OF Alm;
END_VAR
VAR CONSTANT
	almNoAlarm : UINT := 0;
END_VAR
VAR
	AlarmBagNotProxLine : UINT := 0;
END_VAR
VAR CONSTANT
	almEmergencyStop : UINT := 1;
END_VAR
VAR
	repRel : UINT := 1;
	repMix : UINT := 2;
END_VAR
VAR CONSTANT
	almMotorOverload : UINT := 2;
	almUldProgFinished : UINT := 3;
	almUldNoBag : UINT := 4;
	almSwitchFault : UINT := 5;
	almBagNotArrived : UINT := 6;
	almBagNotSettled : UINT := 7;
	almBagNotReleased : UINT := 9;
	almLoadNotDropped : UINT := 10;
	almCarriageMoveFault : UINT := 11;
	almPhotocellBlocked : UINT := 12;
	almPhotocellNotMade : UINT := 13;
	almStationNotClosed : UINT := 14;
	almGeneralSequence : UINT := 15;
	almBagNotAtProx : UINT := 16;
	almBagNotShownOnScreen : UINT := 17;
	almInverterFault : UINT := 18;
	almDestinationNotValid : UINT := 19;
	almBagDataError : UINT := 20;
	almBagOverWeight : UINT := 21;
	almStationNotEmpty : UINT := 22;
	almClearingBeltPleaseWait : UINT := 23;
	almSystemStopped : UINT := 25;
	almReleaseSwitchFault : UINT := 26;
	almReceiveSwitchFault : UINT := 27;
	almRailNotAligned : UINT := 28;
	almLiftRefNotFound : UINT := 29;
	almLiftParameterError : UINT := 30;
	almLiftRefSwitchFault : UINT := 31;
	almRotateRefNotFound : UINT := 32;
	almRotateParameterError : UINT := 33;
	almRotateRefSwitchFault : UINT := 34;
	almNoBatchIDfromSQLserver : UINT := 40;
	almAirPressureLow : UINT := 41;
	almSafetyLoading : UINT := 42;
	almSafetyHighLevel : UINT := 43;
	almSafetyVC : UINT := 44;
	almDisableSequence : UINT := 45;
	almBackUpNotRunning : UINT := 50;
	ALM_SERVO_HOIST : UINT := 65;
END_VAR
```

### Alarm.typ
```iecst
(*Insert your comment here.*)

TYPE
	Alm : 	STRUCT
		On : BOOL;
		Bag : UINT;
		ET : TIME;
		InList : BOOL;
		Name : UINT;
		Extra : UINT;
		Beacon : BOOL;
		Time : UDINT;
	END_STRUCT;
END_TYPE
```

### Package Logical/GlobalVariables/Bag - Bag Variables

### Bag.var
```iecst
VAR RETAIN
	Bag : ARRAY[0..MAX_BAGS] OF Bag_typ;
	pBag : UDINT;
END_VAR
VAR CONSTANT
	MAX_BAGS : UINT := 499;
END_VAR
(*CONSTANTS*)
VAR CONSTANT
	CAT_EMPTY_BAG : UDINT := 999; (**Category code for Empty bag*)
	CAT_MIXED_LINEN : UDINT := 998; (**Category code for mixed linen*)
	CAT_MIXED_GARMENTS : UDINT := 997; (**Category code for mixed garments (Ullmer)*)
END_VAR
```

### Bag.typ
```iecst
TYPE
	Bag_typ : 	STRUCT
		Prg : USINT; (*Program*)
		Dst : USINT; (*Destination - Only Supertrack*)
		Wgt : UINT; (*Weight*)
		Cnt : UINT; (*Count (Items)*)
		Ur1 : UINT; (*User 1*)
		Bid : UDINT; (*Bag ID - Supertrack ID*)
		Cat : UDINT; (*Category*)
		Mis : UDINT; (*Batch ID - MIS Mis Server*)
		Cus : UDINT; (*Customer *)
		Ur2 : UDINT; (*User 2*)
		Timestamp : DATE_AND_TIME;
	END_STRUCT;
END_TYPE
```

### Package Logical/GlobalVariables/Data - Data Variables

### Data.var
```iecst
VAR RETAIN
	pMCN : UDINT;
	C : ARRAY[0..99] OF UINT;
	D : ARRAY[0..7999] OF UINT;
	D32 : ARRAY[0..999] OF UDINT;
	pC : UDINT;
	pD : UDINT;
	pD32 : UDINT;
	pRB_Posn : UDINT;
END_VAR
```

### Package Logical/GlobalVariables/Enable - Sequence Request & Enable Variables

### Enable.var
```iecst
VAR
	VCiLock : ARRAY[0..9] OF VCiLock_Posn_Typ;
	EnableRel : Enable_Vars;
	Enable : Enable_Vars;
	RequestRel : Enable_Vars;
	Request : Enable_Vars;
END_VAR
```

### Enable.typ
```iecst
TYPE
	VCiLock_Signals_Type : 	STRUCT
		ReqRelease : BOOL; (*Output [Releasing] - Request to release a bag*)
		EnabRelease : BOOL; (*Input [Releasing] - Enable bag release*)
		InPosn : BOOL; (*Output [Receive] - Carriage in position*)
		ReqSend : BOOL; (*Input [Receive] - Request to send a bag*)
		EnabSend : BOOL; (*Output  [Receive] - Enable sending a bag*)
		ReqPosn : BOOL; (*Input - Request go to a position*)
	END_STRUCT;
	Enable_Vars : 	STRUCT
		Search : UINT;
		TransferBelt : ARRAY[0..4]OF BOOL;
		Ongoing : ARRAY[0..4]OF BOOL;
		Offgoing : ARRAY[0..4]OF BOOL;
		BSN : ARRAY[0..4]OF BOOL;
		BSF : ARRAY[0..9]OF BOOL;
		FB : ARRAY[0..4]OF BOOL;
		IC : ARRAY[0..9]OF BOOL;
		DC : ARRAY[0..9]OF BOOL;
		LU : ARRAY[0..9]OF BOOL;
		PI : ARRAY[0..9]OF BOOL;
		PC : ARRAY[0..9]OF BOOL;
		PN : ARRAY[0..99]OF BOOL;
		PF : ARRAY[0..9]OF BOOL;
		SB : ARRAY[0..9]OF BOOL;
		SK : ARRAY[0..9]OF BOOL;
		SP : ARRAY[0..39]OF BOOL;
		VC : ARRAY[0..9]OF BOOL;
		WB : ARRAY[0..4]OF BOOL;
		SDP : ARRAY[0..2]OF BOOL;
		FDC : ARRAY[0..2]OF BOOL;
		FDCEmpty : ARRAY[0..2]OF BOOL;
		SDC1Drop : BOOL;
		DCEmptyRelease : ARRAY[0..10]OF BOOL;
		EmptyBagInSVC : ARRAY[0..5]OF BOOL;
		SVC1LowLevel : BOOL;
		SVC3LowLevel : BOOL;
		SVC3HighLevel : BOOL;
		SVC2FullBagLowLevel : BOOL;
		SVC2AtTop : BOOL;
		SVC4ToSDP1 : BOOL;
		SVCFullBag : ARRAY[0..4]OF BOOL;
		VC_LowLevel : ARRAY[0..4]OF BOOL;
		SVCEmptyBag : ARRAY[0..4]OF BOOL;
		VC_HighLevel : ARRAY[0..4]OF BOOL;
	END_STRUCT;
	VCiLock_Posn_Typ : 	STRUCT
		Posn : ARRAY[0..5]OF VCiLock_Signals_Type;
	END_STRUCT;
END_TYPE
```

### Package Logical/GlobalVariables/IO - IO Variables

### IO.var
```iecst
VAR
	WeightRaw : ARRAY[0..99] OF Wieght_typ;
	AI261Raw : ARRAY[0..19] OF DINT;
	AI1223 : ARRAY[0..17] OF INT := [18(0)];
	OK : ARRAY[0..450] OF BOOL;
	StnOK : ARRAY[0..128] OF BOOL;
	X : ARRAY[0..399] OF CardInputs;
	Y : ARRAY[0..399] OF CardOutputs;
	YForceDisable : ARRAY[0..399] OF CardOutputs;
END_VAR
```

### IO.typ
```iecst
TYPE
	CardInputs : 	STRUCT
		X01 : BOOL;
		X02 : BOOL;
		X03 : BOOL;
		X04 : BOOL;
		X05 : BOOL;
		X06 : BOOL;
		X07 : BOOL;
		X08 : BOOL;
		X09 : BOOL;
		X10 : BOOL;
		X11 : BOOL;
		X12 : BOOL;
		X13 : BOOL;
		X14 : BOOL;
		X15 : BOOL;
		X16 : BOOL;
	END_STRUCT;
	CardOutputs : 	STRUCT
		Y01 : BOOL;
		Y02 : BOOL;
		Y03 : BOOL;
		Y04 : BOOL;
		Y05 : BOOL;
		Y06 : BOOL;
		Y07 : BOOL;
		Y08 : BOOL;
		Y09 : BOOL;
		Y10 : BOOL;
		Y11 : BOOL;
		Y12 : BOOL;
		Y13 : BOOL;
		Y14 : BOOL;
		Y15 : BOOL;
		Y16 : BOOL;
	END_STRUCT;
	Wieght_typ : 	STRUCT
		Wgt_Channel_1 : DINT;
		Wgt_Channel_2 : DINT;
		Config_Channel_1 : USINT;
		Config_Channel_2 : USINT;
	END_STRUCT;
END_TYPE
```

### Package Logical/GlobalVariables/Line - Line Status Variables

### Line.var
```iecst
VAR RETAIN
	Line : ARRAY[0..99] OF Line_Typ;
END_VAR
```

### Line.typ
```iecst
TYPE
	Line_Typ : 	STRUCT
		Clear : BOOL;
		Full : BOOL;
		Trip : BOOL;
		FirstBag : UINT;
		LastBag : UINT;
		Space : UINT;
		SpaceBIT : UINT;
	END_STRUCT;
END_TYPE
```

### Package Logical/GlobalVariables/Loading - Loading [Sorting Station] Variables

### Loading.var
```iecst
VAR
	StnPrev : ARRAY[0..60] OF Bag_typ;
	Ldg : ARRAY[0..4] OF Loading_Vars;
	Stn : ARRAY[0..60] OF Stn_Vars;
END_VAR
VAR CONSTANT
	MAX_WEIGHSTATIONS : UINT := 14;
END_VAR
VAR
	AI351RAW_01 : INT;
	AI351RAW_02 : INT;
END_VAR
```

### Loading.typ
```iecst
TYPE
	Loading_Vars : 	STRUCT
		EnableStnRelease : BOOL;
		BeltHasRun : BOOL;
		Found : UINT;
		Line : UINT;
		Search : UINT;
		Stations : ARRAY[0..MAX_WEIGHSTATIONS]OF USINT;
		NoStations : USINT;
	END_STRUCT;
	Stn_Vars : 	STRUCT
		DestManual : UINT;
		LampOn : BOOL;
		GreenLamp : BOOL;
		QTime : UINT;
		ReleaseButton : BOOL;
		SpacesRequired : UINT;
		SP1 : BOOL;
		SP2 : BOOL;
		SP3 : BOOL;
		Count : UINT;
		Closed : BOOL;
		CloseFlap : BOOL;
		CntInput : BOOL;
		Weight : INT;
		Open : BOOL;
		MixCustomer : BOOL;
		PBCount : UINT;
		Purge : BOOL;
		Unlock : BOOL;
		ManualRelease : BOOL;
		PurgeReverse : BOOL;
	END_STRUCT;
END_TYPE
```

### Library Logical/GlobalVariables/Loading/Ldg_Funct (IEC)

#### Ldg_Funct.fun - Exported functions and function blocks
```iecst
FUNCTION LDG_GetBagFromStation : UINT (**Get the bag number from the station number*) (*$GROUP=User,$CAT=User,$GROUPICON=User.png,$CATICON=User.png*)
	VAR_INPUT
		StationBagsStart : UINT;
		StationNum : UINT;
	END_VAR
END_FUNCTION

FUNCTION LDG_GetStationFromBag : UINT (**Get the station number from bag*) (*$GROUP=User,$CAT=User,$GROUPICON=User.png,$CATICON=User.png*)
	VAR_INPUT
		StationBagsStart : UINT; (**Bag number that the stations start at*)
		BagNum : UINT; (** Bag number for station to calculate*)
	END_VAR
END_FUNCTION
```

#### LDG_GetBagFromStation.st
```iecst
(* *Get the bag number from the station number *)
FUNCTION LDG_GetBagFromStation

	LDG_GetBagFromStation := StationBagsStart + StationNum - 1;

END_FUNCTION
```

#### LDG_GetStationFromBag.ab
```automation-basic
(* *Get the station number from bag *)
FUNCTION LDG_GetStationFromBag
	IF BagNum >= StationBagsStart THEN
		LDG_GetStationFromBag :=  BagNum - StationBagsStart + 1
	ELSE
		LDG_GetStationFromBag := 0;
		ENDIF;
END_FUNCTION
```

### Machine.typ - Global data types
```iecst
(********************************************************************
 * COPYRIGHT --
 ********************************************************************
 * Package: TrackView
 * File: TrackView.typ
 * Author: Administrator
 * Created: March 02, 2009
 ********************************************************************
 * Data types of package TrackView
 ********************************************************************)

TYPE
	Typ_MachineStatus : 	STRUCT
		MACHINE_NO : UDINT; (*MACHINE NUMBER 6 - DIGITS*)
		DATA_VALID : USINT; (*0 - OFFLINE / 1 - ONLINE*)
		MACHINE_STATUS : USINT; (*0 - OFF ; 1 - ON WITHOUT MESSAGE ; 2 - ON WITH MESSAGE *)
		MSG_TYPE : USINT; (*0 - WITHOUT MESSAGE ; 1 - WARNING ; 2 - ALARM*)
		SPARE_FREI_1 : USINT; (*NOT USED*)
		MSG_NR : UINT; (*0 - NO MESSAGE ; >0 - WARNING OR ALARM*)
		SPARE_FREI_2 : UINT; (*NOT USED*)
	END_STRUCT;
END_TYPE
```

### Machine.var - Global variables
```iecst
(********************************************************************
 * COPYRIGHT --
 ********************************************************************
 * Package: TrackView
 * File: TrackView.var
 * Author: Dave Jefferys
 * Created: March 02, 2009
 ********************************************************************
 * Variables of package TrackView
 ********************************************************************)
VAR
	MCN : ARRAY[0..99] OF Typ_MachineStatus := [100(0)]; (*Machine Status*)
END_VAR
```

### Package Logical/GlobalVariables/Std - Standard Variables

### Standard.var
```iecst
VAR
	SafetyPLC_Ok : BOOL;
END_VAR
VAR CONSTANT
	MAX_DESTINATIONS : USINT := 99;
END_VAR
VAR
	VCStatus : ARRAY[0..9] OF UINT := [10(0)];
	Std : Std_Vars;
	Test : Test_Vars;
	DestCountStorage : ARRAY[0..MAX_DESTINATIONS] OF UINT; (*Count of each destiantion code in storage*)
	DestCountSystem : ARRAY[0..MAX_DESTINATIONS] OF UINT; (*Count of each destination code in the system*)
	DestCountArea1 : ARRAY[0..MAX_DESTINATIONS] OF UINT; (*Count of each destination in a selected area*)
	DestCountArea2 : ARRAY[0..MAX_DESTINATIONS] OF UINT; (*Count of each destination in a selected area*)
	DestCountArea3 : ARRAY[0..MAX_DESTINATIONS] OF UINT; (*Count of each destination in a selected area*)
	AutomaticLineAllocation : BOOL;
	AutoLineAllocation : BOOL;
	BidStn : UDINT;
	pnlStatusMessage : ARRAY[0..29] OF STRING[20];
	pnlStatus : ARRAY[0..19] OF UINT;
	pnlName : ARRAY[0..29] OF STRING[25];
	DoorOpen : ARRAY[0..49] OF TIME;
	EasiSortHasRun : ARRAY[0..20] OF TIME;
	StationClose : ARRAY[0..20] OF BOOL;
	LongestTime : ARRAY[0..99] OF UINT;
	DebugMode : BOOL;
	Indication : ARRAY[0..79] OF BOOL;
	TestSystem : BOOL;
END_VAR
```

### Standard.typ
```iecst
TYPE
	WriteDisplay : 	STRUCT
		Data : ARRAY[0..7]OF USINT;
	END_STRUCT;
	Test_Vars : 	STRUCT
		TransferBelt : BOOL;
		Stations : BOOL;
		Dischargers : BOOL;
	END_STRUCT;
	Std_Vars : 	STRUCT
		HaltSys : BOOL;
		HaltSysZone : ARRAY[0..4]OF BOOL;
		StopSystem : BOOL;
		SafetyOnZone : ARRAY[0..4]OF BOOL;
		SafetyOn : BOOL;
		AutoMaticRelease : BOOL;
		AutoRecirculation : BOOL;
		AutoLineAllocation : BOOL;
		BagsWithDestinations : BOOL;
		BagsWithDestinations2 : BOOL;
		BagWithDestAtFront : BOOL;
		BagSpacing : USINT;
		Clock100ms : BOOL;
		Clock200ms : BOOL;
		Clock500ms : BOOL;
		Clock1s : BOOL;
		Clock2s : BOOL;
		EStop : BOOL;
		EStopLoading : BOOL;
		EnableOverUnderRelease : BOOL;
		MaxAreas : UINT;
		MaxProg : USINT;
		MaxCats : UDINT;
		MaxCust : UDINT;
		MaxDischargers : USINT;
		MaxIO : UINT;
		MaxLines : UINT;
		MaxLinesBuffers : UINT;
		MaxWeighstations : UINT;
		MaxCountingStations : UINT;
		MaxStationBanks : UINT;
		MaxSearch : UINT;
		MinReleaseWeight : UINT;
		Monitor : UINT;
		MotorOverload : BOOL;
		MotorOverloadLoading : BOOL;
		PairingLoop : BOOL;
		Purging : BOOL;
		PurgeCompleted : BOOL;
		RepSpacing : USINT;
		StnBatchCode : UINT;
		StnsInQ : BOOL;
		StnsToPurge : ARRAY[0..4]OF BOOL;
		StationBagsStart : UINT;
		StationBagDisplay : UINT;
		CountingBagsStart : UINT;
		StationReports : BOOL;
		StationsClosed : BOOL;
		UnloadingMaxDepth : UINT;
		CustomerFIFO : BOOL;
		CustomerFound : BOOL;
		CustomerNewFound : BOOL;
		CustomerEditFound : BOOL;
		PLCStn : USINT;
		MaxSeq : USINT;
		PLCStnString : STRING[1];
		ReversingBelt : BOOL;
		PurgeBank : ARRAY[0..4]OF PurgeBatch_typ;
		AutoPurge : BOOL;
		MinPurgeWeight : USINT;
		StationBankReg : UINT;
		Drives_AllowLocalMode : BOOL;
	END_STRUCT;
	ReadDisplay : 	STRUCT
		Data : ARRAY[0..7]OF USINT;
	END_STRUCT;
	PurgeBatch_typ : 	STRUCT
		PurgeBatch : ARRAY[0..98]OF UINT;
		PurgeBagQty : UINT;
		PurgeBatchCount : UINT;
		PurgeBatchWieght : UINT;
		PurgeOn : UINT;
		StationsStatus : ARRAY[0..1]OF UDINT;
	END_STRUCT;
	fiLOCAL_OBJ : 	STRUCT
		StateMan : UINT;
		ErrMan : UINT;
		Init : UDINT;
	END_STRUCT;
	comstype : 	STRUCT
		delime : UINT;
		delim : ARRAY[0..1]OF USINT;
		tx_cnt : UINT;
		rx_cnt : UINT;
		tx_len : UINT;
		rx_len : UINT;
		argc : UINT;
		argv : UDINT;
		idle : UINT;
	END_STRUCT;
END_TYPE
```

### Package Logical/GlobalVariables/Unloading - Unloading Program Variables

### Unloading.var
```iecst
VAR RETAIN
	Uld : ARRAY[0..20] OF Uld_Vars;
END_VAR
```

### Unloading.typ
```iecst
TYPE
	Uld_Vars : 	STRUCT
		SDCReady : BOOL;
		SDCSpaces : UINT;
		DischargerStartLine : UINT;
		LastCustQtyComplete : UINT;
		FIFOCustomer : UDINT;
		FIFOCustomerFound : BOOL;
		FIFONextCustomer : UDINT;
	END_STRUCT;
END_TYPE
```

### Package Logical/GlobalVariables/BatchID - Batch ID Variables

### BatchID.var
```iecst
VAR
	BatchID : ARRAY[0..9] OF UDINT;
	BatchIDStatus : UDINT;
	RunningWithoutMISServer : BOOL;
END_VAR
VAR CONSTANT
	StatusNotUsed : UDINT := 0;
	StatusOnline : UDINT := 1;
	StatusOffline : UDINT := 2;
	StatusRunIfNoConnection : UDINT := 4;
END_VAR
```

### Package Logical/GlobalVariables/CustomerChange - A package of related programs and data objects.

### CustomerChange.typ - Global data types
```iecst
(********************************************************************
 * COPYRIGHT -- HP
 ********************************************************************
 * Package: CustomerChange
 * File: CustomerChange.typ
 * Author: treamsbottom
 * Created: November 26, 2014
 ********************************************************************
 * Data types of package CustomerChange
 ********************************************************************)

TYPE
	CustChangeDisp_Typ : 	STRUCT
		Message : STRING[32];
		MessageText_Colour : UINT;
		InputLock : UINT;
		InputText_Colour : UINT;
		New_CustomerNo : UDINT;
	END_STRUCT;
END_TYPE
```

### CustomerChange.var - Global variables
```iecst
(********************************************************************
 * COPYRIGHT -- HP
 ********************************************************************
 * Package: CustomerChange
 * File: CustomerChange.var
 * Author: treamsbottom
 * Created: November 26, 2014
 ********************************************************************
 * Variables of package CustomerChange
 ********************************************************************)
VAR
	CustomerChangeDisplay : ARRAY[0..9] OF CustChangeDisp_Typ;
END_VAR
```

### Global.var
```iecst
VAR
	SVC1RequestEmpty : BOOL;
	EnableSDC2Empty : BOOL;
	SVC1Status : UINT;
END_VAR
```

### Package Logical/Documents - Documents

- Base PLC Program Versions.doc (binary file, 31744 bytes)
### Package Logical/Sequences - *

### Package Logical/Sequences/10ms - 10ms Tasks

### Package Logical/Sequences/10ms/Scan - Scan Time Variables

### Scan.typ
```iecst
TYPE
	ScanTime : 	STRUCT
		Start : TIME;
		End : TIME;
		Time : UINT;
		Min : UINT;
		Max : UINT;
	END_STRUCT;
END_TYPE
```

### Scan.var
```iecst
VAR
	TCScan : ARRAY[0..8] OF ScanTime;
END_VAR
```

- Program Logical/Sequences/10ms/Scan/zzTC2str (IEC) - * TC2 Start - Scan Time Calculation (no source held here)

- Program Logical/Sequences/10ms/Scan/zzTC2end (IEC) - * TC2 End - Scan Time Calculation (no source held here)

### Program Logical/Sequences/10ms/zzStd (IEC) - * Standard Functions

#### zzstd.ab
```automation-basic
;Version 1.00 First Issue
;Version 2.00 Added Bag[0] and Removed Mitsubishi M90xx's clock's
;Version 3.00 24/06/2009 New Bag 32bit etc.. D.J.

PROGRAM _INIT

;Memory Address Pointers

;Note - pC was mem_adr_C in old programs
pC			= ADR(C)
pD			= ADR(D)
pD32		= ADR(D32)
pBag		= ADR(Bag)
pRB_Posn	= ADR(RB_Posn)
pMCN		= ADR(MCN)

END_PROGRAM

PROGRAM _CYCLIC

;Set all of bag 0 to Zero for use when deleting bags
Bag[0].Prg 		= 0
Bag[0].Dst 		= 0
Bag[0].Wgt 		= 0
Bag[0].Cus 		= 0
Bag[0].Cat		= 0
Bag[0].Mis 		= 0
Bag[0].Cnt 		= 0
Bag[0].Bid		= 0

;Standard Clocks
TimerClkPT[0] = 5 	;100ms
TimerClkPT[1] = 10 	;200ms
TimerClkPT[2] = 25 	;500ms
TimerClkPT[3] = 50 	;1s
TimerClkPT[4] = 100 ;2s

LOOP n = 0 TO 4 DO

	TimerClkA[n].IN = NOT TimerClkB[n].Q
	TimerClkA[n].PT = TimerClkPT[n]
	TimerClkA[n] FUB TON_10ms()

	TimerClkB[n].IN = TimerClkA[n].Q
	TimerClkB[n].PT = TimerClkPT[n]
	TimerClkB[n] FUB TON_10ms()

ENDLOOP

Std.Clock100ms 	= TimerClkA[0].Q
Std.Clock200ms 	= TimerClkA[1].Q ;M9031
Std.Clock500ms 	= TimerClkA[2].Q
Std.Clock1s 	= TimerClkA[3].Q ;M9032
Std.Clock2s 	= TimerClkA[4].Q ;M9033
END_PROGRAM
```

### Program Logical/Sequences/10ms/zzConst (IEC) - * System Constants - Adjust to Suit

#### zzconst.var
```iecst
VAR
	n : USINT;
	x : USINT;
END_VAR
```

#### zzconst.ab
```automation-basic
;------------------------------------------------
;Version 1.00 01/05/2001 D.J. First Issue
;Version 2.00 24/06/2009 D.J. 32bit Added MaxProg
;------------------------------------------------

PROGRAM _INIT

Std.MaxSeq = 49
Std.PLCStn = 0
itoa(Std.PLCStn,ADR(Std.PLCStnString))

Std.AutoLineAllocation	= FALSE		;Use Automatic Line Allocation?

Std.AutoMaticRelease   	= TRUE		;Set to TRUE for AutoMatic Release using setpoints. FALSE for Push-Button Release
Std.StationReports  	= TRUE 		;Transfer reports to PC

Std.PairingLoop   		= FALSE
Std.CustomerFIFO		= TRUE		;Use Customer FIFO Table

Std.MaxIO				= 39		;Max PLC I/O Cards - check X and Y array size

Std.AutoPurge 			= TRUE

Std.MaxProg				= 99		;Max Program / Classification (Old Category) - Should be 99 or less Max = 255
Std.MaxCats           	= 99		;Max Categories
Std.MaxCust           	= 99		;Max Customers
Std.MaxDischargers    	= 9			;Total Dischargers
Std.MaxLines          	= 17		;Max Storage Lines
Std.MaxAreas			= 11			;Max Storage Areas
Std.MaxLinesBuffers   	= 49		;Storage lines + Buffers
Std.MaxWeighstations  	= MAX_WEIGHSTATIONS			;Total Weighstations
Std.MaxStationBanks		= 2 		;Total Banks of sorting Stations
Std.MaxSearch			= 1   		;Include all station banks and Loading VC's etc

Std.MinReleaseWeight  	= 30		;Include 10ths
Std.MinPurgeWeight		= 15;10

Std.StationBagsStart	= 201		;Bag Number of first bank of sorting stations
Std.StationBagDisplay 	= 201		;Bag Number of second bank of sorting stations

Std.StationBankReg 		= 0 ; Start of D reg where releasing station is stored + 900 i.e to use 901 for bank 1 set to 0.

//SET MAX_WEIGHSTATIONS

Ldg[1].NoStations = 7
LOOP n = 1 TO Ldg[1].NoStations DO
	Ldg[1].Stations[n]	= n
ENDLOOP

;;Stns 2-22 even numbers
Ldg[2].NoStations = 14
;x = 1
LOOP x = 8 TO Ldg[2].NoStations DO
;	IF (n MOD 2 = 0) THEN // Even Number
		Ldg[2].Stations[x]		= x
;		INC x
;	ENDIF
ENDLOOP

Ldg[3].NoStations 	= 0
Ldg[3].Stations[1]	= 0

Ldg[4].NoStations 	= 0
Ldg[4].Stations[1]	= 0

;Enter the First and Last bag for all the Storage lines including buffers
Line[1].FirstBag = 1
Line[1].LastBag  = 6

Line[2].FirstBag = 7
Line[2].LastBag  = 12

Line[3].FirstBag = 13
Line[3].LastBag  = 18

Line[4].FirstBag = 19
Line[4].LastBag  = 24

Line[5].FirstBag = 25
Line[5].LastBag  = 30

Line[6].FirstBag = 31
Line[6].LastBag  = 36

Line[7].FirstBag = 0
Line[7].LastBag  = 0

Line[8].FirstBag = 0
Line[8].LastBag  = 0

Line[9].FirstBag = 110
Line[9].LastBag  = 118 ; BUFFER AFTER CLU1\2

	Line[10].FirstBag = 0
	Line[10].LastBag  = 0

	Line[11].FirstBag = 51
	Line[11].LastBag  = 55

	Line[12].FirstBag = 61
	Line[12].LastBag  = 65

	Line[13].FirstBag = 71 ;SVC 4 High level buffer
	Line[13].LastBag  = 73

	Line[14].FirstBag = 77
	Line[14].LastBag  = 79

	Line[15].FirstBag = 81
	Line[15].LastBag  = 82

	Line[16].FirstBag = 86
	Line[16].LastBag  = 87

	Line[17].FirstBag = 91
	Line[17].LastBag  = 92 ;Pair loop

	Line[18].FirstBag = 96
	Line[18].LastBag  = 97

	Line[19].FirstBag = 101 ;Pair loop
	Line[19].LastBag  = 102 ;Pair loop

	Line[20].FirstBag = 136
	Line[20].LastBag  = 144

	Line[21].FirstBag = 0
	Line[21].LastBag  = 0

	Line[22].FirstBag = 0
	Line[22].LastBag  = 0

	Line[23].FirstBag = 123 ;SVC 4 Low level buffer
	Line[23].LastBag  = 134

	Line[24].FirstBag = 146
	Line[24].LastBag  = 149

	Line[25].FirstBag = 0
	Line[25].LastBag  = 0

	Line[26].FirstBag = 0
	Line[26].LastBag  = 0

	Line[27].FirstBag = 0
	Line[27].LastBag  = 0

	Line[28].FirstBag = 0
	Line[28].LastBag  = 0

	Line[29].FirstBag = 0
	Line[29].LastBag  = 0

	Line[30].FirstBag = 301
	Line[30].LastBag  = 308
;	Line[31].FirstBag = 261
;Line[31].LastBag  = 261

;Line[32].FirstBag = 231
;Line[32].LastBag  = 231

;Line[33].FirstBag = 229
;Line[33].LastBag  = 229

;Line[34].FirstBag = 226
;Line[34].LastBag  = 227

END_PROGRAM

PROGRAM _CYCLIC

Std.EnableOverUnderRelease = FALSE ;X6C 	;Override KeySwitch - See Stn_Q
Bag[0]
;Storage Area transfer to TrackView
D[250] = Std.MaxAreas
;Ensure reply is sent to trackview for Weigh calib to stop mutilpe writes to sql
IF (Std.MaxWeighstations = 0) THEN
	IF (D32[230] >= 0) THEN
		D32[231] = D32[230]
	ELSE
		D32[230] = 1
	ENDIF
ENDIF
END_PROGRAM
```

### Program Logical/Sequences/10ms/zzTrip (IEC) - * Counting Trips with debounce

#### zztrip.var
```iecst
VAR
	CountOld : ARRAY[0..59] OF UINT;
	TripPLS : ARRAY[0..59] OF R_TRIG;
	Timer : ARRAY[0..59] OF TON_10ms;
	CountTrip : ARRAY[0..59] OF BOOL;
	n : UINT;
	Start : BOOL;
END_VAR
```

#### zztrip.ab
```automation-basic
PROGRAM _CYCLIC

;--------------
;Counting trips
;--------------

CountTrip[1]  = X[4].X01;Line1
CountTrip[2]  = X[4].X02
CountTrip[3]  = X[4].X03
CountTrip[4]  = X[4].X04
CountTrip[5]  = X[4].X05
CountTrip[6]  = X[4].X06
CountTrip[7]  = X[4].X07
CountTrip[8]  = X[4].X08
CountTrip[9]  = X[3].X12  ;full bags out CLU1&2
CountTrip[10] = X[8].X11
CountTrip[11] = X[4].X15;line11

CountTrip[12] = X[4].X13 ;SP2 buffer
CountTrip[13] = X[9].X06 ;offgoing buffer high level
CountTrip[14] = X[4].X11
CountTrip[15] = X[1].X01 ;SVC 2 Fullbag out high level
CountTrip[16] = X[1].X07 ;SLU1 Full bag out
CountTrip[17] = X[1].X13
CountTrip[18] = X[2].X03    ; NEEDS INPUT
CountTrip[19] = X[2].X09    ; NEEDS INPUT
CountTrip[20] = X[4].X09
CountTrip[21] = X[9].X01   ;CPC1 Buffer
CountTrip[22] = X[3].X16
CountTrip[23] = X[8].X13 ;offgoing buffer low level
CountTrip[24] = X[4].X12 ;sic 2 bag out at top
CountTrip[25] = X[10].X10
CountTrip[26] = X[10].X11
CountTrip[27] = X[7].X13 ;svc 2 full bag out low level
CountTrip[28] = X[10].X16 ;svc 3 full bag out low level
CountTrip[29] = X[11].X04 ;slu1 empty bag buffer
CountTrip[30] = X[7].X07 ;sic 2 bag out at top
CountTrip[31] = X[2].X12
CountTrip[32] = X[1].X04 ;????????????????????????????????????????????
CountTrip[33] = X[6].X11 ;CDC1 BAG OUT
CountTrip[34] = X[6].X07
CountTrip[35] = X[8].X14
CountTrip[36] = X[8].X15
CountTrip[37] = X[10].X06
CountTrip[38] = X[8].X02
CountTrip[39] = X[9].X13
CountTrip[40] = X[11].X09
CountTrip[41] = X[10].X03
CountTrip[42] = X[6].X15
CountTrip[43] = X[9].X04
CountTrip[44] = X[8].X07
CountTrip[45] = X[7].X03
CountTrip[46] = X[6].X04
CountTrip[47] = X[5].X16

LOOP n = 1 TO Std.MaxLinesBuffers DO
	IF Start THEN
		C[n] = 2
		D[900 + n] := 1;
	ENDIF

	TripPLS[n].CLK = CountTrip[n]
	TripPLS[n] FUB R_TRIG()

	IF TripPLS[n].Q AND Timer[n].Q AND (C[n] < 2) THEN
		C[n] = C[n] + 1
	ENDIF

	Timer[n].IN = NOT CountTrip[n]
	Timer[n].PT = 20;100 = 1second
	Timer[n] FUB TON_10ms()

	Line[n].Full 	= (C[n] = 1)
	Line[n].Clear 	= ((C[n] >= 2) AND Timer[n].Q)

	Line[n].Trip	= (((CountOld[n] <> C[n]) AND (C[n] <> 0)) OR CountTrip[n]) ;Use for Bag Arrived at destination
	CountOld[n] 	= C[n]

ENDLOOP
Start = FALSE
END_PROGRAM
```

### Program Logical/Sequences/10ms/zzBagID (IEC, version 3.00.0) - Bag ID Allocation

#### zzBagID.var - Local variables
```iecst
(********************************************************************
 * COPYRIGHT --
 ********************************************************************
 * Program: zzBagID
 * File: zzBagID.var
 * Author: Dave
 * Created: September 26, 2010
 ********************************************************************
 * Local variables of program zzBagID
 ********************************************************************)
VAR
	n : UINT;
	BagByteSize : UDINT;
	NoOfBags : UDINT;
END_VAR
```

#### zzBagID.ab - Cyclic code
```automation-basic
(********************************************************************
 * COPYRIGHT --
 ********************************************************************
 * Program: zzBagID
 * File: zzBagID.ab
 * Author: Dave
 * Created: September 26, 2010
 ********************************************************************
 * Implementation of program zzBagID
 ********************************************************************)

;Version 2.00 03/11/2011 D.J. Added Check if already allocated as now only between 1000 and 32000
;Version 3.00 14/05/2012 D.J. Changed to UDINT - range now from 1000 to Hex FFFFFFFF

PROGRAM _CYCLIC

	;Bag ID number allocation from 1000 to Hex FFFFFFFF if below then wait for TrackView to send the correct value

	;Allocate station bag ID next bag ID for use
	IF ((BidStn = 0) AND (D32[200] >= 1000)) THEN

		;Keep within range UDINT
		;IF (D32[200] > $FFFFFFFF) THEN
		IF (D32[200] > 32000) THEN
			D32[200] = 1000
		ENDIF

		BidStn 		= D32[200]
		D32[200] 	= (D32[200] + 1)

		;Check if new allocated ID is still used if so then clear

		BagByteSize = SIZEOF(Bag[0])
		NoOfBags = (SIZEOF(Bag)/BagByteSize) - 1 ; - 1 to set to 0 based index
		LOOP n = 1 TO UINT(NoOfBags) DO
			IF Bag[n].Bid = BidStn THEN
				BidStn = 0
			ENDIF
		EXITIF BidStn = 0
		ENDLOOP

	ENDIF

END_PROGRAM
```

### Program Logical/Sequences/10ms/zzBatchID (IEC, version 1.10.0) - Batch ID from MIS SQL Server

#### zzBatchID.var - Local variables
```iecst
(********************************************************************
 * COPYRIGHT --
 ********************************************************************
 * Program: zzSLQid
 * File: zzSLQid.var
 * Author: Dave
 * Created: July 08, 2011
 ********************************************************************
 * Local variables of program zzSLQid
 ********************************************************************)
VAR
	MachID : UDINT;
	LocationNumber : UDINT;
	ElementIndex : UDINT;
	IDRecieved : BOOL;
	STEP : UINT;
	StnBag : UINT;
	n : UINT;
	Bank : UINT;
	FoundIndex : UINT;
	FoundBag : UINT;
	BatchNumber : UDINT;
	ReplyID : UDINT;
	RequestID : BOOL;
	WaitReply : BOOL;
	MaxBags : UINT;
	PLCiD : UDINT;
	ServerStatus : UDINT;
	TON_MISstatus : TON_10ms;
	StateOffline : BOOL;
	StateRunWithout : BOOL;
	StateNotUsed : BOOL;
	StatusNotUse : BOOL;
	StateOnline : BOOL;
	TON_MISonline : TON_10ms;
END_VAR
```

#### zzBatchID.ab - Implementation code
```automation-basic
;------------------------------------------------------------------
;zzBatchid - Get batch number from TrackView (Provided by MIS Server)
;------------------------------------------------------------------

;Version 1.00 02/11/2011 D.J. First Issue
;Version 1.10 02/03/2012 D.J. Changed StateNotUsed	= (BatchIDStatus = 0)

PROGRAM _CYCLIC

	MachID 			= 999001 ;Set Required Machine Number
	BatchNumber		= D32[210]
	ReplyID			= D32[211]

	;If not waiting for a reply from TrackView and BatchID has been cleared
	IF NOT WaitReply THEN

		IF (BatchID[2] = 0) THEN
			LocationNumber 	= 2 		;Location ie Sorting Stations = 1, Transfer Belt = 2, Loading VC = 3
			ElementIndex 	= 0 		;Element Index 0 = First Index
			WaitReply		= TRUE
		ELSE IF (BatchID[3] = 0) THEN
			LocationNumber 	= 3 		;Location ie Sorting Stations = 1, Transfer Belt = 2, Loading VC = 3
			ElementIndex 	= 0 		;Element Index 0 = First Index
			WaitReply		= TRUE
		ENDIF

		IF WaitReply THEN
			PLCiD			= PLCiD + 1
			IF (PLCiD > 32000) THEN
				PLCiD = 1
			ENDIF
			D32[212] = PLCiD
			D32[213] = MachID
			D32[214] = LocationNumber
			D32[215] = ElementIndex
			D32[216] = 0 ;Time Stamp Not Used
		ENDIF

	ENDIF

	;Wait for TrackView to reply with a Batch ID (Number)
	IF (WaitReply AND (ReplyID = PLCiD)) THEN
		IF (LocationNumber > 0) AND (LocationNumber <= SIZEOF(BatchID)) THEN
			BatchID[LocationNumber]	= BatchNumber
		ENDIF
		WaitReply 	= FALSE
		D32[212] 	= 0
		D32[213] 	= 0
		D32[214] 	= 0
		D32[215] 	= 0
		D32[216] 	= 0 ;Time Stamp Not Used
	ENDIF

	;Set Status for Mis server connection - allow running with no connection if option selected in TrackView

	;Online is only considered after 10 seconds delay as TrackView will set the status to online to re-try connection
	TON_MISstatus.IN = (BatchIDStatus <> D32[217])
	TON_MISstatus.PT = 500
	TON_MISstatus FUB TON_10ms()

	IF TON_MISstatus.Q THEN
		BatchIDStatus 	= D32[217] ;Mis Server Status to/from TrackView
	ENDIF

	StateNotUsed	= (BatchIDStatus = 0)
	StateOnline 	= BOOL(BatchIDStatus AND StatusOnline)
	StateOffline 	= BOOL(BatchIDStatus AND StatusOffline)
	StateRunWithout = BOOL(BatchIDStatus AND StatusRunIfNoConnection)

	TON_MISonline.IN = (StateOffline AND StateRunWithout)
	TON_MISonline.PT = 6000
	TON_MISonline FUB TON_10ms()

	RunningWithoutMISServer = (StateNotUsed OR TON_MISonline.Q)

	;-------------------------------------------
	;Sorting Station Batch ID allocation - Fixed
	;-------------------------------------------

	LOOP n = 1 TO Std.MaxWeighstations DO
		StnBag = n + (Std.StationBagsStart[1] - 1) ;Assumes all station bags will follow in order
		Bag[StnBag].Mis = n
	ENDLOOP

END_PROGRAM
```

### Program Logical/Sequences/10ms/zzEditBag (IEC, version 4.00.0) - Bag Data Editing Control

#### zzEditBag.var - Local variables
```iecst
(********************************************************************
 * COPYRIGHT --
 ********************************************************************
 * Program: zzEditBag
 * File: zzEditBag.var
 * Author: Dave
 * Created: September 25, 2010
 ********************************************************************
 * Local variables of program zzEditBag
 ********************************************************************)
VAR CONSTANT
	accOperator : USINT := 0;
	accSupervisor : USINT := 1;
	accEngineer : USINT := 2;
	accProgrammer : USINT := 3;
	accDesigner : USINT := 4;
END_VAR
VAR
	EditPrg : USINT;
	EditCat : UDINT;
	EditCus : UDINT;
	EditWgt : UINT;
	EditCnt : UINT;
	EditDst : USINT;
	EditBid : UDINT;
	EditPosnNow : UDINT;
	EditPosnNew : UDINT;
	EditMode : UDINT;
	EditAccLev : USINT;
	EditStatus : UDINT;
	MaxBags : UINT;
	n : INT;
	BagsToSearch : UINT;
	SearchBag : UINT;
	CatValid : BOOL;
	PrgValid : BOOL;
	CusValid : BOOL;
	EditMis : UDINT;
	EditUr2 : UDINT;
	EditUr1 : UINT;
	BagSize : UINT;
	EditTimeStamp : DATE_AND_TIME;
END_VAR
```

#### zzEditBag.ab - Cyclic code
```automation-basic
(********************************************************************
 * COPYRIGHT --
 ********************************************************************
 * Program: zzEditBag
 * File: zzEditBag.ab
 * Author: Dave
 * Created: September 25, 2010
 ********************************************************************
 * Implementation of program zzEditBag
 ********************************************************************)

;Version 2.00 08/07/2011 D.J. Removed the need to have a Bag ID (Batch Number) for Mis Server compatibility.
;Version 3.00 03/11/2011 D.J. Mis BatchID and BagID now seperated
;Veriosn 4.00 14/05/2012 D.J. New Bag Data Type

PROGRAM _CYCLIC

	EditPrg = USINT(D32[501])
	EditDst	= USINT(D32[502])
	EditWgt = UINT(D32[503])
	EditCnt = UINT(D32[504])
	EditUr1 = UINT(D32[505])
	EditBid = D32[506]
	EditCat = D32[507]
	EditMis = D32[508]
	EditCus	= D32[509]
	EditUr2 = D32[510]
	EditTimeStamp = DT(D32[511])

	EditPosnNow = D32[515]
	EditPosnNew = D32[516]
	EditMode	= D32[517]
	EditAccLev	= USINT(D32[518])
	EditStatus	= D32[519]

	;Loop through all bags 100 per scan and check if ID matches - access > supervisor
	BagSize = SIZEOF(Bag[0])
	MaxBags = ((SIZEOF(Bag) / BagSize) - 1)

	IF (EditStatus = 1) THEN
		EditStatus = 2 ;Searching
	ENDIF

	;Search 100 bags per scan
	LOOP SearchBag = 1 TO MaxBags DO
		;Bag with correct ID found then update
		IF (EditStatus = 2) THEN
			IF ((Bag[SearchBag].Bid = EditBid) AND (Bag[SearchBag].Bid > 0)) THEN
				Bag[SearchBag].Prg 	= EditPrg
				Bag[SearchBag].Dst 	= EditDst
				Bag[SearchBag].Wgt 	= EditWgt
				Bag[SearchBag].Cnt 	= EditCnt
				Bag[SearchBag].Ur1 	= EditUr1

				Bag[SearchBag].Cat 	= EditCat
				Bag[SearchBag].Mis 	= EditMis
				Bag[SearchBag].Cus 	= EditCus
				Bag[SearchBag].Ur2 	= EditUr2
				Bag[SearchBag].Timestamp = EditTimeStamp

				EditStatus 			= 3 ;Complete
			ENDIF
		ENDIF
	ENDLOOP

	;Bag not found and access >= engineer then add bag direct
	IF (EditStatus = 2) THEN
		IF (EditBid > 0) THEN
			IF (EditAccLev >= accSupervisor) AND (EditPosnNew <= MaxBags) THEN
				Bag[EditPosnNew].Prg 	= EditPrg
				Bag[EditPosnNew].Dst 	= EditDst
				Bag[EditPosnNew].Wgt 	= EditWgt
				Bag[EditPosnNew].Cnt 	= EditCnt
				Bag[EditPosnNew].Ur1 	= EditUr1
				Bag[EditPosnNew].Bid 	= EditBid
				Bag[EditPosnNew].Cat 	= EditCat
				Bag[EditPosnNew].Mis 	= EditMis
				Bag[EditPosnNew].Cus 	= EditCus
				Bag[EditPosnNew].Ur2 	= EditUr2
				Bag[EditPosnNew].Timestamp 	= EditTimeStamp
				EditStatus 				= 3 ;Complete
			ELSE
				EditStatus 				= 4 ;Failed
			ENDIF
		ENDIF
	ENDIF
	;Cancel when all bags have been searched
	IF (EditStatus >= 3) THEN
		D32[519] = 0
	ENDIF

END_PROGRAM
```

### Program Logical/Sequences/10ms/zzForceI (IEC)

#### zzforcei.var
```iecst
VAR
	n : UINT;
	XForce : CardInputs;
	XForceVal : CardInputs;
	Force : UINT;
	myForceState : UINT;
	myForceValue : UINT;
	myForceCard : UINT;
END_VAR
```

#### zzforcei.ab
```automation-basic
PROGRAM _CYCLIC

;---------------------------
;Input forcing from Graphics
;---------------------------

;Version 1.00 14/09/2006 D.J. First Issue
;Version 2.00 20/11/2009 D.J. Changed to 8 I/O inputs per card  - added upto 4 force cards

LOOP Force = 1 TO 4 DO

	n = ((Force - 1) * 5)

	myForceCard 	= D[380 + n]
	myForceState 	= D[381 + n]
	myForceValue 	= D[382 + n]

	IF (myForceCard > Std.MaxIO) THEN
		myForceCard = 0
	ENDIF

	XForce.X01 		= BIT_TST(myForceState,0)
	XForce.X02 		= BIT_TST(myForceState,1)
	XForce.X03 		= BIT_TST(myForceState,2)
	XForce.X04 		= BIT_TST(myForceState,3)
	XForce.X05 		= BIT_TST(myForceState,4)
	XForce.X06 		= BIT_TST(myForceState,5)
	XForce.X07 		= BIT_TST(myForceState,6)
	XForce.X08 		= BIT_TST(myForceState,7)
	XForce.X09 		= BIT_TST(myForceState,8)
	XForce.X10 		= BIT_TST(myForceState,9)
	XForce.X11 		= BIT_TST(myForceState,10)
	XForce.X12 		= BIT_TST(myForceState,11)
	XForce.X13 		= BIT_TST(myForceState,12)
	XForce.X14 		= BIT_TST(myForceState,13)
	XForce.X15 		= BIT_TST(myForceState,14)
	XForce.X16 		= BIT_TST(myForceState,15)

	XForceVal.X01 	= BIT_TST(myForceValue,0)
	XForceVal.X02 	= BIT_TST(myForceValue,1)
	XForceVal.X03 	= BIT_TST(myForceValue,2)
	XForceVal.X04 	= BIT_TST(myForceValue,3)
	XForceVal.X05 	= BIT_TST(myForceValue,4)
	XForceVal.X06 	= BIT_TST(myForceValue,5)
	XForceVal.X07 	= BIT_TST(myForceValue,6)
	XForceVal.X08 	= BIT_TST(myForceValue,7)
	XForceVal.X09 	= BIT_TST(myForceValue,8)
	XForceVal.X10 	= BIT_TST(myForceValue,9)
	XForceVal.X11 	= BIT_TST(myForceValue,10)
	XForceVal.X12 	= BIT_TST(myForceValue,11)
	XForceVal.X13 	= BIT_TST(myForceValue,12)
	XForceVal.X14 	= BIT_TST(myForceValue,13)
	XForceVal.X15 	= BIT_TST(myForceValue,14)
	XForceVal.X16 	= BIT_TST(myForceValue,15)

	X[myForceCard].X01 = (X[myForceCard].X01 AND NOT XForce.X01) OR (XForce.X01 AND XForceVal.X01)
	X[myForceCard].X02 = (X[myForceCard].X02 AND NOT XForce.X02) OR (XForce.X02 AND XForceVal.X02)
	X[myForceCard].X03 = (X[myForceCard].X03 AND NOT XForce.X03) OR (XForce.X03 AND XForceVal.X03)
	X[myForceCard].X04 = (X[myForceCard].X04 AND NOT XForce.X04) OR (XForce.X04 AND XForceVal.X04)
	X[myForceCard].X05 = (X[myForceCard].X05 AND NOT XForce.X05) OR (XForce.X05 AND XForceVal.X05)
	X[myForceCard].X06 = (X[myForceCard].X06 AND NOT XForce.X06) OR (XForce.X06 AND XForceVal.X06)
	X[myForceCard].X07 = (X[myForceCard].X07 AND NOT XForce.X07) OR (XForce.X07 AND XForceVal.X07)
	X[myForceCard].X08 = (X[myForceCard].X08 AND NOT XForce.X08) OR (XForce.X08 AND XForceVal.X08)
	X[myForceCard].X09 = (X[myForceCard].X09 AND NOT XForce.X09) OR (XForce.X09 AND XForceVal.X09)
	X[myForceCard].X10 = (X[myForceCard].X10 AND NOT XForce.X10) OR (XForce.X10 AND XForceVal.X10)
	X[myForceCard].X11 = (X[myForceCard].X11 AND NOT XForce.X11) OR (XForce.X11 AND XForceVal.X11)
	X[myForceCard].X12 = (X[myForceCard].X12 AND NOT XForce.X12) OR (XForce.X12 AND XForceVal.X12)
	X[myForceCard].X13 = (X[myForceCard].X13 AND NOT XForce.X13) OR (XForce.X13 AND XForceVal.X13)
	X[myForceCard].X14 = (X[myForceCard].X14 AND NOT XForce.X14) OR (XForce.X14 AND XForceVal.X14)
	X[myForceCard].X15 = (X[myForceCard].X15 AND NOT XForce.X15) OR (XForce.X15 AND XForceVal.X15)
	X[myForceCard].X16 = (X[myForceCard].X16 AND NOT XForce.X16) OR (XForce.X16 AND XForceVal.X16)

ENDLOOP

END_PROGRAM
```

### Program Logical/Sequences/10ms/zzBagShuffle (IEC) - * Bag Shuffle including Buffers - Using 'Bag' 

#### zzbagsfl.var
```iecst
VAR RETAIN
	CurrentBag : UINT;
	CurrentLine : UINT;
	LineSp : UINT;
END_VAR
VAR
	NextBag : UINT;
	CurrentDst : UINT;
	BelowMaxLines : BOOL;
	n : UINT;
END_VAR
```
